C09144=1205.549,-72.595,-39.498,179.562,5.497,149.096
C09145=1205.554,-72.845,-39.488,179.559,5.497,149.096
C09146=1205.559,-73.095,-39.476,179.557,5.497,149.097
C09147=1205.565,-73.344,-39.465,179.555,5.497,149.098
C09148=1205.570,-73.594,-39.454,179.553,5.497,149.098
C09149=1205.574,-73.844,-39.443,179.550,5.496,149.099
C09150=1205.580,-74.093,-39.432,179.548,5.497,149.100
C09151=1205.585,-74.343,-39.421,179.545,5.496,149.100
C09152=1205.590,-74.593,-39.410,179.543,5.496,149.101
C09153=1205.596,-74.863,-39.398,179.540,5.496,149.102
C09154=1205.602,-75.134,-39.386,179.538,5.496,149.102
C09155=1205.608,-75.405,-39.373,179.535,5.495,149.103
C09156=1205.613,-75.675,-39.362,179.533,5.496,149.104
C09157=1205.619,-75.925,-39.351,179.530,5.495,149.105
C09158=1205.624,-76.174,-39.340,179.528,5.495,149.105
C09159=1205.629,-76.424,-39.329,179.526,5.495,149.106
C09160=1205.634,-76.674,-39.318,179.523,5.494,149.106
C09161=1205.640,-76.923,-39.307,179.521,5.495,149.107
C09162=1205.645,-77.174,-39.296,179.519,5.494,149.108
C09163=1205.650,-77.423,-39.285,179.516,5.495,149.109
C09164=1205.655,-77.673,-39.275,179.514,5.494,149.109
C09165=1205.661,-77.923,-39.263,179.512,5.494,149.110
C09166=1205.666,-78.172,-39.252,179.510,5.494,149.111
C09167=1205.671,-78.422,-39.241,179.507,5.493,149.111
C09168=1205.676,-78.672,-39.230,179.505,5.494,149.112
C09169=1205.681,-78.921,-39.220,179.502,5.493,149.113
C09170=1205.687,-79.171,-39.208,179.501,5.493,149.113
C09171=1205.692,-79.421,-39.198,179.498,5.493,149.114
C09172=1205.697,-79.670,-39.186,179.496,5.493,149.115
C09173=1205.702,-79.921,-39.176,179.493,5.493,149.115
C09174=1205.707,-80.169,-39.165,179.490,5.492,149.116
C09175=1205.712,-80.420,-39.154,179.489,5.492,149.116
C09176=1205.718,-80.669,-39.143,179.486,5.492,149.117
C09177=1205.723,-80.919,-39.132,179.484,5.492,149.118
C09178=1205.728,-81.169,-39.122,179.481,5.492,149.119
C09179=1205.733,-81.418,-39.111,179.479,5.492,149.119
C09180=1205.738,-81.669,-39.100,179.477,5.491,149.120
C09181=1205.744,-81.918,-39.089,179.475,5.492,149.120
C09182=1205.749,-82.168,-39.079,179.472,5.491,149.121
C09183=1205.755,-82.417,-39.067,179.470,5.491,149.122
C09184=1205.760,-82.667,-39.056,179.468,5.491,149.123
C09185=1205.765,-82.917,-39.046,179.465,5.490,149.123
C09186=1205.770,-83.166,-39.035,179.463,5.491,149.124
C09187=1205.775,-83.417,-39.024,179.461,5.490,149.124
C09188=1205.780,-83.666,-39.013,179.459,5.491,149.125
C09189=1205.785,-83.916,-39.003,179.456,5.490,149.126
C09190=1205.791,-84.165,-38.993,179.454,5.489,149.126
C09191=1205.796,-84.415,-38.981,179.452,5.490,149.127
C09192=1205.801,-84.665,-38.971,179.449,5.489,149.128
C09193=1205.806,-84.914,-38.960,179.447,5.490,149.129
C09194=1205.812,-85.164,-38.950,179.444,5.489,149.129
C09195=1205.817,-85.414,-38.939,179.443,5.489,149.130
C09196=1205.823,-85.663,-38.928,179.440,5.489,149.130
C09197=1205.828,-85.913,-38.917,179.438,5.489,149.131
C09198=1205.833,-86.163,-38.907,179.435,5.489,149.132
C09199=1205.838,-86.413,-38.895,179.433,5.489,149.133
C09200=1205.843,-86.662,-38.885,179.431,5.488,149.133
C09201=1205.848,-86.912,-38.875,179.428,5.488,149.134
C09202=1205.854,-87.162,-38.864,179.426,5.488,149.134
C09203=1205.859,-87.412,-38.853,179.423,5.488,149.135
C09204=1205.864,-87.661,-38.843,179.421,5.488,149.136
C09205=1205.869,-87.911,-38.832,179.419,5.487,149.136
C09206=1205.875,-88.160,-38.821,179.417,5.488,149.137
C09207=1205.880,-88.411,-38.811,179.414,5.487,149.138
C09208=1205.885,-88.660,-38.801,179.412,5.488,149.138
C09209=1205.890,-88.910,-38.790,179.410,5.487,149.139
C09210=1205.895,-89.159,-38.779,179.408,5.487,149.140
C09211=1205.900,-89.409,-38.769,179.405,5.487,149.140
C09212=1205.906,-89.659,-38.758,179.403,5.486,149.141
C09213=1205.911,-89.909,-38.748,179.401,5.487,149.142
C09214=1205.917,-90.159,-38.738,179.398,5.486,149.143
C09215=1205.921,-90.408,-38.726,179.396,5.486,149.143
C09216=1205.927,-90.658,-38.716,179.394,5.486,149.144
C09217=1205.932,-90.908,-38.706,179.392,5.486,149.144
C09218=1205.937,-91.157,-38.696,179.389,5.486,149.145
C09219=1205.942,-91.407,-38.686,179.387,5.486,149.146
C09220=1205.947,-91.657,-38.675,179.385,5.485,149.146
C09221=1205.953,-91.906,-38.664,179.383,5.486,149.147
C09222=1205.958,-92.156,-38.654,179.380,5.485,149.148
C09223=1205.963,-92.406,-38.643,179.378,5.486,149.148
C09224=1205.968,-92.656,-38.633,179.376,5.485,149.149
C09225=1205.974,-92.906,-38.623,179.374,5.485,149.150
C09226=1205.980,-93.155,-38.612,179.371,5.485,149.150
C09227=1205.985,-93.406,-38.602,179.368,5.485,149.151
C09228=1205.990,-93.654,-38.591,179.367,5.485,149.152
C09229=1205.995,-93.905,-38.580,179.364,5.484,149.152
C09230=1206.000,-94.154,-38.571,179.362,5.484,149.153
C09231=1206.005,-94.403,-38.561,179.359,5.484,149.154
C09232=1206.010,-94.654,-38.550,179.357,5.484,149.154
C09233=1206.016,-94.903,-38.540,179.355,5.484,149.155
C09234=1206.021,-95.154,-38.529,179.353,5.484,149.156
C09235=1206.026,-95.403,-38.519,179.350,5.484,149.156
C09236=1206.032,-95.653,-38.509,179.348,5.484,149.157
C09237=1206.037,-95.903,-38.498,179.346,5.483,149.158
C09238=1206.042,-96.152,-38.489,179.344,5.484,149.158
C09239=1206.048,-96.402,-38.478,179.341,5.483,149.159
C09240=1206.053,-96.652,-38.468,179.339,5.484,149.160
C09241=1206.058,-96.901,-38.458,179.337,5.483,149.160
C09242=1206.063,-97.152,-38.447,179.335,5.483,149.161
C09243=1206.069,-97.401,-38.437,179.332,5.483,149.162
C09244=1206.074,-97.650,-38.427,179.330,5.483,149.162
C09245=1206.079,-97.901,-38.417,179.328,5.482,149.163
C09246=1206.084,-98.150,-38.406,179.325,5.482,149.163
C09247=1206.090,-98.400,-38.396,179.323,5.482,149.164
C09248=1206.095,-98.650,-38.386,179.320,5.482,149.165
C09249=1206.100,-98.900,-38.375,179.319,5.482,149.165
C09250=1206.105,-99.149,-38.366,179.316,5.481,149.166
C09251=1206.110,-99.399,-38.355,179.314,5.482,149.167
C09252=1206.116,-99.649,-38.345,179.311,5.481,149.168
C09253=1206.121,-99.898,-38.335,179.309,5.482,149.168
C09254=1206.126,-100.148,-38.325,179.307,5.481,149.169
C09255=1206.131,-100.398,-38.315,179.305,5.481,149.169
C09256=1206.137,-100.647,-38.304,179.302,5.481,149.170
C09257=1206.142,-100.918,-38.294,179.300,5.481,149.171
C09258=1206.148,-101.190,-38.282,179.297,5.481,149.172
C09259=1206.154,-101.461,-38.271,179.295,5.480,149.172
C09260=1206.160,-101.733,-38.261,179.293,5.481,149.173
C09261=1206.164,-101.983,-38.251,179.291,5.480,149.173
C09262=1206.170,-102.232,-38.240,179.288,5.480,149.174
C09263=1206.175,-102.482,-38.230,179.286,5.480,149.175
C09264=1206.180,-102.731,-38.221,179.284,5.480,149.176
C09265=1206.185,-102.981,-38.210,179.281,5.480,149.176
C09266=1206.191,-103.231,-38.200,179.279,5.480,149.177
C09267=1206.196,-103.480,-38.190,179.277,5.480,149.178
C09268=1206.201,-103.731,-38.180,179.275,5.480,149.178
C09269=1206.207,-103.981,-38.170,179.272,5.479,149.179
C09270=1206.212,-104.230,-38.160,179.270,5.480,149.179
C09271=1206.217,-104.479,-38.150,179.268,5.479,149.180
C09272=1206.222,-104.730,-38.140,179.266,5.479,149.181
C09273=1206.228,-104.980,-38.130,179.263,5.479,149.181
C09274=1206.233,-105.229,-38.121,179.261,5.479,149.182
C09275=1206.238,-105.478,-38.110,179.259,5.479,149.183
C09276=1206.243,-105.729,-38.100,179.257,5.479,149.183
C09277=1206.248,-105.978,-38.090,179.254,5.478,149.184
C09278=1206.254,-106.228,-38.081,179.252,5.479,149.185
C09279=1206.260,-106.478,-38.071,179.250,5.478,149.185
C09280=1206.264,-106.728,-38.061,179.248,5.479,149.186
C09281=1206.270,-106.977,-38.050,179.245,5.478,149.187
C09282=1206.276,-107.227,-38.041,179.243,5.478,149.187
C09283=1206.280,-107.477,-38.031,179.241,5.478,149.188
C09284=1206.285,-107.727,-38.021,179.239,5.478,149.189
C09285=1206.290,-107.976,-38.011,179.236,5.477,149.189
C09286=1206.296,-108.226,-38.002,179.234,5.478,149.190
C09287=1206.302,-108.476,-37.991,179.232,5.477,149.191
C09288=1206.307,-108.725,-37.982,179.230,5.477,149.191
C09289=1206.312,-108.976,-37.972,179.227,5.477,149.192
C09290=1206.317,-109.225,-37.962,179.225,5.477,149.193
C09291=1206.322,-109.475,-37.952,179.222,5.477,149.193
C09292=1206.328,-109.724,-37.942,179.221,5.477,149.194
C09293=1206.333,-109.974,-37.933,179.218,5.477,149.194
C09294=1206.338,-110.224,-37.922,179.216,5.477,149.195
C09295=1206.343,-110.473,-37.913,179.214,5.476,149.196
C09296=1206.349,-110.724,-37.903,179.212,5.476,149.196
C09297=1206.355,-110.973,-37.893,179.209,5.476,149.197
C09298=1206.359,-111.222,-37.883,179.207,5.476,149.198
C09299=1206.365,-111.473,-37.874,179.205,5.476,149.198
C09300=1206.370,-111.722,-37.864,179.203,5.476,149.199
C09301=1206.376,-111.973,-37.854,179.200,5.476,149.200
C09302=1206.380,-112.222,-37.845,179.199,5.476,149.200
C09303=1206.386,-112.471,-37.835,179.196,5.475,149.201
C09304=1206.391,-112.721,-37.826,179.194,5.476,149.202
C09305=1206.396,-112.972,-37.815,179.192,5.475,149.202
C09306=1206.401,-113.221,-37.806,179.189,5.475,149.203
C09307=1206.407,-113.471,-37.796,179.187,5.475,149.204
C09308=1206.412,-113.720,-37.786,179.185,5.475,149.204
C09309=1206.418,-113.970,-37.777,179.182,5.474,149.205
C09310=1206.423,-114.220,-37.767,179.180,5.475,149.205
C09311=1206.428,-114.470,-37.758,179.178,5.475,149.206
C09312=1206.433,-114.720,-37.748,179.176,5.474,149.207
C09313=1206.439,-114.970,-37.738,179.174,5.475,149.207
C09314=1206.443,-115.219,-37.729,179.171,5.474,149.208
C09315=1206.449,-115.469,-37.719,179.169,5.475,149.209
C09316=1206.454,-115.718,-37.710,179.167,5.474,149.209
C09317=1206.460,-115.969,-37.700,179.165,5.474,149.210
C09318=1206.465,-116.218,-37.691,179.162,5.474,149.211
C09319=1206.471,-116.468,-37.681,179.161,5.474,149.211
C09320=1206.476,-116.717,-37.671,179.158,5.474,149.212
C09321=1206.481,-116.968,-37.662,179.156,5.474,149.213
C09322=1206.486,-117.217,-37.652,179.154,5.473,149.213
C09323=1206.492,-117.467,-37.642,179.152,5.474,149.214
C09324=1206.497,-117.717,-37.633,179.149,5.473,149.215
C09325=1206.502,-117.967,-37.624,179.147,5.473,149.215
C09326=1206.507,-118.216,-37.614,179.145,5.473,149.216
C09327=1206.513,-118.466,-37.605,179.143,5.473,149.217
C09328=1206.518,-118.716,-37.595,179.140,5.472,149.217
C09329=1206.523,-118.965,-37.586,179.138,5.473,149.218
C09330=1206.528,-119.215,-37.576,179.136,5.472,149.218
C09331=1206.534,-119.465,-37.567,179.134,5.473,149.219
C09332=1206.539,-119.715,-37.557,179.132,5.473,149.220
C09333=1206.544,-119.965,-37.547,179.129,5.472,149.220
C09334=1206.549,-120.215,-37.538,179.127,5.473,149.221
C09335=1206.554,-120.464,-37.529,179.125,5.472,149.222
C09336=1206.560,-120.714,-37.519,179.123,5.472,149.222
C09337=1206.565,-120.964,-37.510,179.120,5.472,149.223
C09338=1206.571,-121.213,-37.500,179.119,5.472,149.223
C09339=1206.576,-121.463,-37.491,179.116,5.472,149.224
C09340=1206.581,-121.713,-37.482,179.114,5.472,149.225
C09341=1206.587,-121.963,-37.472,179.112,5.471,149.225
C09342=1206.592,-122.213,-37.463,179.110,5.472,149.226
C09343=1206.597,-122.462,-37.454,179.107,5.471,149.227
C09344=1206.603,-122.712,-37.444,179.105,5.471,149.227
C09345=1206.608,-122.962,-37.435,179.103,5.471,149.228
C09346=1206.613,-123.211,-37.426,179.101,5.471,149.229
C09347=1206.619,-123.461,-37.416,179.099,5.471,149.229
C09348=1206.624,-123.711,-37.407,179.096,5.471,149.230
C09349=1206.629,-123.960,-37.398,179.094,5.471,149.231
C09350=1206.635,-124.210,-37.388,179.092,5.470,149.231
C09351=1206.640,-124.460,-37.379,179.090,5.471,149.232
C09352=1206.645,-124.710,-37.370,179.087,5.470,149.233
C09353=1206.650,-124.959,-37.361,179.086,5.470,149.233
C09354=1206.656,-125.210,-37.351,179.083,5.470,149.234
C09355=1206.661,-125.459,-37.342,179.081,5.470,149.234
C09356=1206.666,-125.709,-37.333,179.079,5.470,149.235
C09357=1206.672,-125.959,-37.323,179.077,5.470,149.236
C09358=1206.677,-126.209,-37.314,179.074,5.469,149.236
C09359=1206.682,-126.459,-37.305,179.072,5.470,149.237
C09360=1206.687,-126.708,-37.296,179.070,5.470,149.238
C09361=1206.266,-126.720,-37.333,179.066,5.473,149.239
C09362=1206.261,-126.470,-37.342,179.068,5.473,149.239
C09363=1206.255,-126.220,-37.352,179.070,5.473,149.238
C09364=1206.250,-125.970,-37.361,179.073,5.473,149.238
C09365=1206.245,-125.721,-37.370,179.074,5.473,149.237
C09366=1206.239,-125.470,-37.380,179.077,5.474,149.236
C09367=1206.234,-125.221,-37.389,179.079,5.473,149.236
C09368=1206.228,-124.971,-37.398,179.081,5.474,149.235
C09369=1206.224,-124.722,-37.407,179.083,5.474,149.234
C09370=1206.218,-124.471,-37.417,179.086,5.474,149.234
C09371=1206.213,-124.222,-37.426,179.088,5.474,149.233
C09372=1206.208,-123.972,-37.435,179.090,5.474,149.233
C09373=1206.202,-123.722,-37.445,179.092,5.474,149.232
C09374=1206.197,-123.472,-37.454,179.095,5.475,149.231
C09375=1206.192,-123.223,-37.463,179.097,5.474,149.231
C09376=1206.186,-122.973,-37.473,179.099,5.474,149.230
C09377=1206.181,-122.723,-37.482,179.101,5.475,149.229
C09378=1206.176,-122.474,-37.491,179.103,5.474,149.229
C09379=1206.170,-122.223,-37.501,179.106,5.475,149.228
C09380=1206.165,-121.973,-37.510,179.107,5.475,149.227
C09381=1206.160,-121.724,-37.520,179.110,5.475,149.227
C09382=1206.155,-121.474,-37.529,179.112,5.475,149.226
C09383=1206.149,-121.224,-37.538,179.114,5.476,149.226
C09384=1206.145,-120.975,-37.548,179.116,5.475,149.225
C09385=1206.139,-120.724,-37.557,179.119,5.476,149.224
C09386=1206.133,-120.475,-37.566,179.121,5.476,149.224
C09387=1206.128,-120.225,-37.576,179.123,5.476,149.223
C09388=1206.123,-119.975,-37.585,179.125,5.476,149.222
C09389=1206.118,-119.726,-37.595,179.128,5.476,149.222
C09390=1206.112,-119.476,-37.604,179.130,5.476,149.221
C09391=1206.107,-119.226,-37.613,179.132,5.476,149.220
C09392=1206.102,-118.977,-37.623,179.134,5.476,149.220
C09393=1206.096,-118.727,-37.632,179.136,5.476,149.219
C09394=1206.091,-118.477,-37.642,179.139,5.476,149.218
C09395=1206.085,-118.227,-37.651,179.140,5.476,149.218
C09396=1206.081,-117.977,-37.661,179.143,5.477,149.217
C09397=1206.075,-117.727,-37.671,179.145,5.476,149.216
C09398=1206.070,-117.478,-37.680,179.147,5.477,149.216
C09399=1206.065,-117.228,-37.689,179.149,5.477,149.215
C09400=1206.059,-116.978,-37.700,179.152,5.477,149.215
C09401=1206.054,-116.729,-37.708,179.154,5.477,149.214
C09402=1206.049,-116.479,-37.719,179.156,5.478,149.213
C09403=1206.044,-116.229,-37.728,179.158,5.477,149.213
C09404=1206.038,-115.980,-37.738,179.161,5.478,149.212
C09405=1206.033,-115.729,-37.747,179.163,5.478,149.211
C09406=1206.028,-115.480,-37.757,179.165,5.478,149.211
C09407=1206.023,-115.230,-37.766,179.167,5.478,149.210
C09408=1206.017,-114.980,-37.776,179.170,5.478,149.209
C09409=1206.012,-114.730,-37.785,179.172,5.478,149.209
C09410=1206.007,-114.481,-37.795,179.174,5.478,149.208
C09411=1206.001,-114.231,-37.804,179.176,5.478,149.208
C09412=1205.996,-113.982,-37.814,179.179,5.479,149.207
C09413=1205.991,-113.731,-37.824,179.181,5.478,149.206
C09414=1205.985,-113.481,-37.834,179.183,5.478,149.205
C09415=1205.980,-113.231,-37.843,179.185,5.479,149.205
C09416=1205.975,-112.982,-37.853,179.187,5.478,149.204
C09417=1205.970,-112.733,-37.863,179.190,5.479,149.204
C09418=1205.964,-112.482,-37.872,179.191,5.479,149.203
C09419=1205.959,-112.233,-37.882,179.194,5.479,149.202
C09420=1205.954,-111.982,-37.892,179.196,5.479,149.202
C09421=1205.949,-111.733,-37.901,179.198,5.480,149.201
C09422=1205.943,-111.484,-37.912,179.200,5.479,149.200
C09423=1205.938,-111.234,-37.920,179.203,5.480,149.200
C09424=1205.932,-110.984,-37.931,179.205,5.479,149.199
C09425=1205.928,-110.735,-37.940,179.207,5.480,149.198
C09426=1205.922,-110.484,-37.950,179.209,5.480,149.198
C09427=1205.917,-110.235,-37.960,179.212,5.480,149.197
C09428=1205.912,-109.985,-37.970,179.214,5.480,149.197
C09429=1205.906,-109.735,-37.979,179.216,5.480,149.196
C09430=1205.901,-109.486,-37.989,179.219,5.480,149.195
C09431=1205.896,-109.236,-38.000,179.221,5.480,149.194
C09432=1205.891,-108.986,-38.009,179.223,5.481,149.194
C09433=1205.885,-108.736,-38.019,179.225,5.481,149.193
C09434=1205.880,-108.487,-38.029,179.228,5.481,149.193
C09435=1205.874,-108.237,-38.038,179.230,5.481,149.192
C09436=1205.869,-107.987,-38.048,179.232,5.481,149.191
C09437=1205.864,-107.737,-38.059,179.235,5.481,149.191
C09438=1205.859,-107.488,-38.068,179.237,5.481,149.190
C09439=1205.853,-107.238,-38.078,179.239,5.482,149.189
C09440=1205.848,-106.989,-38.087,179.241,5.481,149.189
C09441=1205.843,-106.738,-38.098,179.244,5.482,149.188
C09442=1205.838,-106.489,-38.108,179.246,5.481,149.187
C09443=1205.832,-106.239,-38.117,179.248,5.482,149.187
C09444=1205.827,-105.989,-38.127,179.250,5.482,149.186
C09445=1205.822,-105.739,-38.138,179.253,5.482,149.185
C09446=1205.817,-105.490,-38.147,179.254,5.482,149.185
C09447=1205.811,-105.240,-38.157,179.257,5.483,149.184
C09448=1205.806,-104.990,-38.167,179.259,5.482,149.183
C09449=1205.801,-104.740,-38.177,179.262,5.483,149.183
C09450=1205.796,-104.491,-38.187,179.263,5.483,149.182
C09451=1205.790,-104.241,-38.198,179.266,5.483,149.182
C09452=1205.786,-103.991,-38.207,179.268,5.483,149.181
C09453=1205.780,-103.741,-38.217,179.271,5.483,149.180
C09454=1205.774,-103.491,-38.227,179.272,5.483,149.180
C09455=1205.769,-103.242,-38.237,179.275,5.484,149.179
C09456=1205.764,-102.992,-38.247,179.277,5.483,149.178
C09457=1205.759,-102.742,-38.258,179.280,5.484,149.177
C09458=1205.754,-102.493,-38.267,179.281,5.484,149.177
C09459=1205.749,-102.242,-38.277,179.284,5.484,149.176
C09460=1205.743,-101.993,-38.287,179.286,5.484,149.176
C09461=1205.737,-101.743,-38.298,179.289,5.484,149.175
C09462=1205.732,-101.472,-38.308,179.291,5.484,149.174
C09463=1205.727,-101.201,-38.319,179.294,5.484,149.173
C09464=1205.721,-100.930,-38.331,179.296,5.484,149.173
C09465=1205.715,-100.658,-38.342,179.298,5.484,149.172
C09466=1205.710,-100.408,-38.351,179.300,5.485,149.172
C09467=1205.705,-100.158,-38.362,179.303,5.484,149.171
C09468=1205.699,-99.909,-38.372,179.305,5.485,149.170
C09469=1205.694,-99.659,-38.381,179.307,5.484,149.169
C09470=1205.689,-99.409,-38.392,179.310,5.485,149.169
C09471=1205.683,-99.160,-38.402,179.312,5.486,149.168
C09472=1205.678,-98.910,-38.412,179.314,5.485,149.167
C09473=1205.674,-98.660,-38.422,179.317,5.486,149.167
C09474=1205.668,-98.410,-38.433,179.319,5.486,149.166
C09475=1205.662,-98.161,-38.443,179.321,5.486,149.166
C09476=1205.657,-97.911,-38.453,179.323,5.486,149.165
C09477=1205.652,-97.661,-38.464,179.326,5.486,149.164
C09478=1205.647,-97.412,-38.473,179.328,5.486,149.164
C09479=1205.642,-97.162,-38.484,179.330,5.487,149.163
C09480=1205.636,-96.912,-38.494,179.332,5.486,149.162
C09481=1205.631,-96.663,-38.504,179.335,5.487,149.162
C09482=1205.626,-96.412,-38.515,179.337,5.487,149.161
C09483=1205.620,-96.163,-38.525,179.339,5.487,149.160
C09484=1205.615,-95.913,-38.536,179.341,5.487,149.160
C09485=1205.610,-95.663,-38.545,179.344,5.487,149.159
C09486=1205.605,-95.414,-38.555,179.346,5.487,149.158
C09487=1205.600,-95.164,-38.566,179.348,5.488,149.158
C09488=1205.594,-94.914,-38.576,179.350,5.487,149.157
C09489=1205.588,-94.664,-38.586,179.353,5.488,149.156
C09490=1205.583,-94.414,-38.597,179.355,5.488,149.156
C09491=1205.578,-94.165,-38.608,179.357,5.488,149.155
C09492=1205.574,-93.915,-38.618,179.359,5.488,149.154
C09493=1205.568,-93.666,-38.628,179.362,5.488,149.154
C09494=1205.563,-93.416,-38.638,179.365,5.488,149.153
C09495=1205.558,-93.166,-38.649,179.366,5.488,149.152
C09496=1205.552,-92.916,-38.659,179.369,5.489,149.152
C09497=1205.547,-92.666,-38.670,179.371,5.489,149.151
C09498=1205.542,-92.417,-38.680,179.374,5.489,149.150
C09499=1205.537,-92.166,-38.690,179.375,5.489,149.150
C09500=1205.531,-91.918,-38.701,179.378,5.489,149.149
C09501=1205.526,-91.668,-38.712,179.380,5.489,149.148
C09502=1205.521,-91.418,-38.722,179.383,5.489,149.148
C09503=1205.515,-91.168,-38.732,179.385,5.489,149.147
C09504=1205.510,-90.918,-38.743,179.387,5.490,149.147
C09505=1205.505,-90.669,-38.753,179.389,5.489,149.146
C09506=1205.501,-90.419,-38.764,179.392,5.490,149.145
C09507=1205.495,-90.170,-38.774,179.395,5.490,149.144
C09508=1205.489,-89.920,-38.784,179.396,5.490,149.144
C09509=1205.484,-89.670,-38.795,179.399,5.491,149.143
C09510=1205.479,-89.421,-38.806,179.401,5.490,149.142
C09511=1205.474,-89.171,-38.816,179.404,5.491,149.142
C09512=1205.468,-88.921,-38.826,179.406,5.490,149.141
C09513=1205.463,-88.671,-38.837,179.408,5.491,149.141
C09514=1205.458,-88.421,-38.847,179.410,5.491,149.140
C09515=1205.453,-88.172,-38.859,179.413,5.491,149.139
C09516=1205.448,-87.922,-38.869,179.415,5.491,149.138
C09517=1205.443,-87.672,-38.879,179.417,5.492,149.138
C09518=1205.437,-87.422,-38.890,179.419,5.491,149.137
C09519=1205.432,-87.173,-38.901,179.422,5.492,149.137
C09520=1205.427,-86.923,-38.911,179.424,5.492,149.136
C09521=1205.422,-86.673,-38.922,179.426,5.492,149.135
C09522=1205.416,-86.424,-38.933,179.429,5.493,149.135
C09523=1205.411,-86.174,-38.943,179.431,5.492,149.134
C09524=1205.406,-85.924,-38.953,179.433,5.493,149.133
C09525=1205.401,-85.675,-38.965,179.435,5.492,149.133
C09526=1205.395,-85.425,-38.975,179.438,5.493,149.132
C09527=1205.390,-85.175,-38.985,179.440,5.493,149.131
C09528=1205.384,-84.926,-38.997,179.442,5.493,149.131
C09529=1205.379,-84.675,-39.008,179.445,5.494,149.130
C09530=1205.374,-84.426,-39.018,179.447,5.493,149.129
C09531=1205.369,-84.176,-39.029,179.450,5.494,149.128
C09532=1205.364,-83.927,-39.039,179.451,5.494,149.128
C09533=1205.359,-83.676,-39.050,179.454,5.494,149.127
C09534=1205.354,-83.427,-39.061,179.456,5.494,149.127
C09535=1205.348,-83.177,-39.071,179.459,5.494,149.126
C09536=1205.344,-82.928,-39.083,179.461,5.494,149.125
C09537=1205.338,-82.678,-39.093,179.463,5.495,149.125
C09538=1205.333,-82.428,-39.103,179.466,5.495,149.124
C09539=1205.328,-82.179,-39.114,179.468,5.495,149.123
C09540=1205.322,-81.928,-39.125,179.471,5.495,149.123
C09541=1205.317,-81.679,-39.136,179.473,5.495,149.122
C09542=1205.312,-81.429,-39.147,179.475,5.496,149.121
C09543=1205.307,-81.179,-39.158,179.477,5.495,149.121
C09544=1205.301,-80.930,-39.168,179.480,5.496,149.120
C09545=1205.296,-80.680,-39.179,179.482,5.495,149.119
C09546=1205.291,-80.431,-39.190,179.484,5.496,149.119
C09547=1205.285,-80.180,-39.201,179.487,5.496,149.118
C09548=1205.280,-79.931,-39.212,179.489,5.496,149.117
C09549=1205.275,-79.681,-39.223,179.491,5.497,149.117
C09550=1205.270,-79.431,-39.234,179.493,5.496,149.116
C09551=1205.265,-79.182,-39.244,179.496,5.497,149.115
C09552=1205.260,-78.932,-39.255,179.498,5.497,149.115
C09553=1205.254,-78.682,-39.266,179.500,5.497,149.114
C09554=1205.249,-78.433,-39.277,179.503,5.497,149.113
C09555=1205.244,-78.183,-39.288,179.505,5.497,149.113
C09556=1205.239,-77.934,-39.299,179.508,5.498,149.112
C09557=1205.234,-77.684,-39.310,179.510,5.497,149.111
C09558=1205.228,-77.434,-39.321,179.512,5.498,149.111
C09559=1205.223,-77.184,-39.332,179.514,5.498,149.110
C09560=1205.218,-76.934,-39.343,179.517,5.498,149.109
C09561=1205.213,-76.685,-39.354,179.519,5.499,149.109
C09562=1205.207,-76.435,-39.365,179.522,5.498,149.108
C09563=1205.202,-76.185,-39.376,179.524,5.499,149.107
C09564=1205.197,-75.936,-39.387,179.526,5.499,149.107
C09565=1205.192,-75.686,-39.398,179.528,5.499,149.106
C09566=1205.186,-75.416,-39.410,179.531,5.499,149.105
C09567=1205.180,-75.145,-39.422,179.533,5.499,149.105
C09568=1205.175,-74.874,-39.434,179.536,5.500,149.104
C09569=1205.169,-74.604,-39.446,179.539,5.500,149.103
C09570=1205.164,-74.354,-39.457,179.541,5.500,149.102
C09571=1205.159,-74.104,-39.468,179.543,5.500,149.102
C09572=1205.153,-73.855,-39.479,179.546,5.500,149.101
C09573=1205.148,-73.605,-39.491,179.548,5.500,149.100
C09574=1205.143,-73.354,-39.501,179.550,5.501,149.100
C09575=1205.138,-73.106,-39.512,179.552,5.501,149.099
C09576=1205.132,-72.856,-39.524,179.555,5.501,149.098
C09577=1205.127,-72.605,-39.535,179.557,5.501,149.098
C09578=1205.122,-72.356,-39.546,179.560,5.501,149.097
C09579=1205.117,-72.107,-39.558,179.562,5.502,149.097
C09580=1205.112,-71.856,-39.568,179.564,5.502,149.096
C09581=1205.107,-71.607,-39.579,179.567,5.502,149.095
C09582=1205.101,-71.357,-39.591,179.569,5.502,149.094
C09583=1205.096,-71.108,-39.602,179.571,5.502,149.094
C09584=1205.091,-70.858,-39.613,179.574,5.502,149.093
C09585=1205.085,-70.608,-39.624,179.576,5.502,149.093
C09586=1205.080,-70.359,-39.636,179.578,5.503,149.092
C09587=1205.075,-70.108,-39.646,179.581,5.503,149.091
C09588=1205.069,-69.859,-39.658,179.583,5.503,149.090
C09589=1205.065,-69.610,-39.669,179.586,5.503,149.090
C09590=1205.060,-69.360,-39.680,179.588,5.503,149.089
C09591=1205.055,-69.110,-39.692,179.590,5.504,149.088
C09592=1205.049,-68.860,-39.702,179.592,5.504,149.088
C09593=1205.044,-68.611,-39.714,179.595,5.504,149.087
C09594=1205.039,-68.361,-39.726,179.598,5.504,149.086
C09595=1205.034,-68.111,-39.737,179.600,5.504,149.086
C09596=1205.028,-67.862,-39.748,179.602,5.504,149.085
C09597=1205.023,-67.612,-39.759,179.604,5.505,149.084
C09598=1205.018,-67.362,-39.771,179.607,5.505,149.084
C09599=1205.013,-67.112,-39.782,179.609,5.505,149.083
C09600=1205.008,-66.863,-39.793,179.611,5.505,149.082
C09601=1205.002,-66.613,-39.805,179.614,5.505,149.082
C09602=1204.998,-66.364,-39.816,179.616,5.505,149.081
C09603=1204.992,-66.114,-39.828,179.618,5.506,149.080
C09604=1204.987,-65.864,-39.838,179.621,5.506,149.080
C09605=1204.981,-65.614,-39.850,179.623,5.506,149.079
C09606=1204.976,-65.365,-39.861,179.626,5.506,149.078
C09607=1204.971,-65.115,-39.873,179.628,5.506,149.078
C09608=1204.966,-64.865,-39.885,179.630,5.507,149.077
C09609=1204.960,-64.616,-39.896,179.633,5.507,149.076
C09610=1204.956,-64.366,-39.907,179.635,5.507,149.076
C09611=1204.950,-64.116,-39.919,179.637,5.507,149.075
C09612=1204.945,-63.867,-39.931,179.639,5.507,149.074
C09613=1204.940,-63.617,-39.943,179.642,5.508,149.074
C09614=1204.935,-63.368,-39.953,179.645,5.508,149.073
C09615=1204.929,-63.117,-39.965,179.646,5.508,149.072
C09616=1204.924,-62.868,-39.976,179.649,5.508,149.072
C09617=1204.919,-62.618,-39.988,179.652,5.509,149.071
C09618=1204.914,-62.368,-39.999,179.654,5.509,149.070
C09619=1204.909,-62.118,-40.011,179.656,5.509,149.070
C09620=1204.903,-61.869,-40.022,179.659,5.509,149.069
C09621=1204.898,-61.619,-40.034,179.661,5.509,149.068
C09622=1204.893,-61.370,-40.045,179.663,5.510,149.068
C09623=1204.888,-61.120,-40.057,179.665,5.510,149.067
C09624=1204.883,-60.870,-40.068,179.668,5.510,149.066
C09625=1204.878,-60.620,-40.080,179.671,5.510,149.066
C09626=1204.873,-60.371,-40.091,179.673,5.510,149.065
C09627=1204.867,-60.121,-40.103,179.676,5.511,149.064
C09628=1204.863,-59.872,-40.115,179.677,5.511,149.064
C09629=1204.857,-59.622,-40.127,179.680,5.511,149.063
C09630=1204.852,-59.372,-40.139,179.683,5.511,149.062
C09631=1204.847,-59.123,-40.150,179.685,5.511,149.062
C09632=1204.842,-58.873,-40.162,179.687,5.512,149.061
C09633=1204.837,-58.623,-40.173,179.690,5.512,149.060
C09634=1204.831,-58.374,-40.185,179.692,5.512,149.060
C09635=1204.826,-58.124,-40.197,179.694,5.512,149.059
C09636=1204.821,-57.874,-40.208,179.696,5.512,149.058
C09637=1204.815,-57.625,-40.220,179.699,5.513,149.058
C09638=1204.811,-57.375,-40.231,179.702,5.513,149.057
C09639=1204.806,-57.126,-40.244,179.704,5.513,149.056
C09640=1204.800,-56.876,-40.256,179.706,5.513,149.056
C09641=1204.796,-56.626,-40.267,179.709,5.514,149.055
C09642=1204.790,-56.376,-40.279,179.711,5.514,149.054
C09643=1204.785,-56.126,-40.291,179.713,5.514,149.054
C09644=1204.780,-55.877,-40.302,179.716,5.514,149.053
C09645=1204.774,-55.627,-40.313,179.718,5.514,149.052
C09646=1204.770,-55.378,-40.325,179.721,5.515,149.052
C09647=1204.764,-55.128,-40.337,179.723,5.515,149.051
C09648=1204.759,-54.878,-40.349,179.725,5.515,149.050
C09649=1204.754,-54.629,-40.360,179.728,5.516,149.050
C09650=1204.749,-54.379,-40.372,179.730,5.515,149.049
C09651=1204.743,-54.130,-40.385,179.732,5.516,149.048
C09652=1204.738,-53.880,-40.397,179.735,5.516,149.048
C09653=1204.733,-53.630,-40.408,179.737,5.516,149.047
C09654=1204.728,-53.380,-40.420,179.740,5.516,149.046
C09655=1204.723,-53.131,-40.433,179.742,5.517,149.046
C09656=1204.718,-52.881,-40.444,179.744,5.517,149.045
C09657=1204.713,-52.631,-40.456,179.747,5.517,149.044
C09658=1204.707,-52.381,-40.468,179.749,5.518,149.044
C09659=1204.703,-52.132,-40.480,179.751,5.517,149.043
C09660=1204.697,-51.882,-40.492,179.754,5.518,149.042
C09661=1204.692,-51.632,-40.503,179.757,5.518,149.041
C09662=1204.687,-51.383,-40.516,179.758,5.518,149.041
C09663=1204.682,-51.133,-40.527,179.761,5.519,149.040
C09664=1204.677,-50.883,-40.539,179.764,5.519,149.040
C09665=1204.671,-50.634,-40.551,179.766,5.519,149.039
C09666=1204.666,-50.384,-40.564,179.768,5.519,149.038
C09667=1204.661,-50.134,-40.576,179.771,5.520,149.037
C09668=1204.656,-49.885,-40.587,179.773,5.519,149.037
C09669=1204.651,-49.635,-40.599,179.775,5.520,149.036
C09670=1204.645,-49.366,-40.612,179.779,5.520,149.035
C09671=1204.640,-49.095,-40.625,179.781,5.520,149.035
C09672=1204.634,-48.825,-40.638,179.783,5.520,149.034
C09673=1204.628,-48.555,-40.651,179.786,5.521,149.033
C09674=1204.623,-48.306,-40.663,179.789,5.521,149.033
C09675=1204.618,-48.056,-40.675,179.790,5.521,149.032
C09676=1204.613,-47.807,-40.688,179.793,5.522,149.031
C09677=1204.607,-47.557,-40.700,179.796,5.522,149.031
C09678=1204.602,-47.307,-40.711,179.798,5.522,149.030
C09679=1204.597,-47.058,-40.724,179.800,5.522,149.029
C09680=1204.592,-46.808,-40.735,179.803,5.523,149.029
C09681=1204.587,-46.559,-40.748,179.805,5.522,149.028
C09682=1204.582,-46.309,-40.760,179.808,5.523,149.027
C09683=1204.577,-46.058,-40.772,179.810,5.524,149.027
C09684=1204.572,-45.809,-40.785,179.812,5.523,149.026
C09685=1204.566,-45.559,-40.797,179.815,5.524,149.025
C09686=1204.561,-45.309,-40.809,179.817,5.524,149.025
C09687=1204.556,-45.060,-40.820,179.819,5.524,149.024
C09688=1204.551,-44.811,-40.833,179.822,5.524,149.023
C09689=1204.546,-44.561,-40.845,179.825,5.525,149.022
C09690=1204.541,-44.311,-40.858,179.827,5.526,149.022
C09691=1204.535,-44.061,-40.869,179.829,5.525,149.021
C09692=1204.530,-43.812,-40.882,179.832,5.526,149.021
C09693=1204.525,-43.562,-40.894,179.834,5.526,149.020
C09694=1204.520,-43.313,-40.907,179.836,5.526,149.019
C09695=1204.514,-43.063,-40.918,179.839,5.526,149.018
C09696=1204.510,-42.813,-40.931,179.842,5.527,149.018
C09697=1204.505,-42.563,-40.944,179.843,5.527,149.017
C09698=1204.499,-42.314,-40.956,179.846,5.527,149.017
C09699=1204.495,-42.065,-40.968,179.849,5.528,149.016
C09700=1204.489,-41.815,-40.980,179.851,5.527,149.015
C09701=1204.484,-41.565,-40.992,179.853,5.528,149.014
C09702=1204.479,-41.315,-41.004,179.856,5.528,149.014
C09703=1204.474,-41.066,-41.017,179.858,5.528,149.013
C09704=1204.468,-40.817,-41.029,179.861,5.528,149.012
C09705=1204.464,-40.566,-41.042,179.863,5.529,149.012
C09706=1204.459,-40.317,-41.054,179.866,5.530,149.011
C09707=1204.453,-40.067,-41.066,179.868,5.529,149.011
C09708=1204.448,-39.818,-41.079,179.870,5.530,149.010
C09709=1204.443,-39.568,-41.091,179.873,5.530,149.009
C09710=1204.437,-39.318,-41.103,179.875,5.530,149.008
C09711=1204.432,-39.069,-41.116,179.878,5.530,149.008
C09712=1204.428,-38.819,-41.129,179.880,5.531,149.007
C09713=1204.422,-38.569,-41.141,179.882,5.531,149.007
C09714=1204.417,-38.320,-41.153,179.885,5.531,149.006
C09715=1204.412,-38.070,-41.166,179.887,5.532,149.005
C09716=1204.407,-37.820,-41.178,179.890,5.532,149.004
C09717=1204.402,-37.571,-41.190,179.892,5.532,149.004
C09718=1204.397,-37.321,-41.203,179.895,5.532,149.003
C09719=1204.392,-37.072,-41.216,179.897,5.533,149.003
C09720=1204.386,-36.821,-41.228,179.899,5.533,149.002
C09721=1204.381,-36.572,-41.241,179.902,5.533,149.001
C09722=1204.375,-36.323,-41.254,179.904,5.534,149.000
C09723=1204.370,-36.074,-41.266,179.906,5.534,149.000
C09724=1204.366,-35.823,-41.279,179.909,5.534,148.999
C09725=1204.360,-35.574,-41.291,179.912,5.534,148.998
C09726=1204.355,-35.324,-41.304,179.914,5.535,148.998
C09727=1204.350,-35.075,-41.316,179.916,5.535,148.997
C09728=1204.345,-34.824,-41.329,179.919,5.535,148.996
C09729=1204.340,-34.575,-41.341,179.921,5.536,148.996
C09730=1204.335,-34.326,-41.354,179.923,5.536,148.995
C09731=1204.329,-34.076,-41.367,179.926,5.536,148.994
C09732=1204.324,-33.827,-41.380,179.929,5.537,148.994
C09733=1204.319,-33.576,-41.392,179.931,5.537,148.993
C09734=1204.314,-33.327,-41.404,179.933,5.537,148.993
C09735=1204.309,-33.077,-41.417,179.936,5.538,148.992
C09736=1204.304,-32.828,-41.430,179.938,5.538,148.991
C09737=1204.299,-32.578,-41.443,179.940,5.538,148.990
C09738=1204.294,-32.329,-41.456,179.943,5.538,148.990
C09739=1204.288,-32.079,-41.468,179.946,5.539,148.989
C09740=1204.283,-31.829,-41.480,179.948,5.539,148.988
C09741=1204.278,-31.579,-41.493,179.950,5.539,148.988
C09742=1204.273,-31.330,-41.506,179.953,5.540,148.987
C09743=1204.268,-31.081,-41.518,179.955,5.540,148.986
C09744=1204.262,-30.831,-41.532,179.958,5.540,148.986
C09745=1204.258,-30.581,-41.545,179.960,5.540,148.985
C09746=1204.253,-30.332,-41.557,179.963,5.541,148.984
C09747=1204.248,-30.082,-41.570,179.965,5.541,148.984
C09748=1204.242,-29.833,-41.582,179.968,5.542,148.983
C09749=1204.237,-29.583,-41.596,179.970,5.542,148.983
C09750=1204.232,-29.333,-41.609,179.972,5.542,148.982
C09751=1204.227,-29.083,-41.620,179.975,5.543,148.981
C09752=1204.222,-28.833,-41.633,179.977,5.542,148.980
C09753=1204.217,-28.584,-41.646,179.980,5.543,148.980
C09754=1204.211,-28.334,-41.659,179.982,5.543,148.979
C09755=1204.207,-28.084,-41.672,179.985,5.544,148.978
C09756=1204.201,-27.835,-41.685,179.987,5.543,148.978
C09757=1204.196,-27.586,-41.697,179.989,5.544,148.977
C09758=1204.191,-27.335,-41.711,179.992,5.545,148.976
C09759=1204.186,-27.086,-41.724,179.995,5.545,148.976
C09760=1204.181,-26.837,-41.736,179.997,5.545,148.975
C09761=1204.176,-26.587,-41.749,179.999,5.545,148.974
C09762=1204.171,-26.338,-41.763,-179.998,5.546,148.974
C09763=1204.166,-26.088,-41.776,-179.995,5.546,148.973
C09764=1204.161,-25.838,-41.789,-179.993,5.546,148.972
C09765=1204.155,-25.589,-41.802,-179.991,5.547,148.972
C09766=1204.150,-25.340,-41.814,-179.988,5.547,148.971
C09767=1204.146,-25.089,-41.827,-179.986,5.548,148.970
C09768=1204.140,-24.840,-41.840,-179.984,5.547,148.970
C09769=1204.135,-24.591,-41.853,-179.981,5.548,148.969
C09770=1204.130,-24.341,-41.866,-179.978,5.548,148.968
C09771=1204.125,-24.091,-41.879,-179.976,5.549,148.968
C09772=1204.119,-23.842,-41.892,-179.974,5.549,148.967
C09773=1204.115,-23.592,-41.905,-179.972,5.549,148.966
C09774=1204.109,-23.323,-41.920,-179.969,5.550,148.966
C09775=1204.104,-23.053,-41.933,-179.966,5.550,148.965
C09776=1204.098,-22.783,-41.947,-179.963,5.550,148.964
C09777=1204.093,-22.514,-41.962,-179.960,5.551,148.963
C09778=1204.087,-22.264,-41.975,-179.958,5.551,148.963
C09779=1204.082,-22.015,-41.988,-179.956,5.551,148.962
C09780=1204.077,-21.765,-42.001,-179.953,5.552,148.962
C09781=1204.072,-21.515,-42.014,-179.951,5.552,148.961
C09782=1204.067,-21.265,-42.027,-179.948,5.553,148.960
C09783=1204.062,-21.016,-42.041,-179.946,5.552,148.960
C09784=1204.057,-20.767,-42.053,-179.943,5.553,148.959
C09785=1204.051,-20.517,-42.067,-179.941,5.553,148.958
C09786=1204.046,-20.267,-42.079,-179.939,5.554,148.958
C09787=1204.042,-20.018,-42.093,-179.937,5.554,148.957
C09788=1204.036,-19.768,-42.106,-179.934,5.554,148.956
C09789=1204.031,-19.519,-42.119,-179.931,5.555,148.956
C09790=1204.026,-19.269,-42.133,-179.929,5.555,148.955
C09791=1204.021,-19.020,-42.146,-179.926,5.556,148.954
C09792=1204.016,-18.770,-42.159,-179.924,5.556,148.953
C09793=1204.010,-18.520,-42.172,-179.921,5.556,148.953
C09794=1204.006,-18.270,-42.185,-179.919,5.557,148.952
C09795=1204.000,-18.021,-42.199,-179.916,5.557,148.952
C09796=1203.996,-17.771,-42.212,-179.914,5.557,148.951
C09797=1203.990,-17.522,-42.225,-179.912,5.557,148.950
C09798=1203.985,-17.273,-42.238,-179.909,5.558,148.950
C09799=1203.980,-17.023,-42.252,-179.906,5.558,148.949
C09800=1203.975,-16.773,-42.265,-179.904,5.559,148.948
C09801=1203.970,-16.524,-42.279,-179.902,5.559,148.948
C09802=1203.965,-16.274,-42.291,-179.899,5.559,148.947
C09803=1203.959,-16.024,-42.305,-179.897,5.560,148.946
C09804=1203.955,-15.775,-42.318,-179.894,5.560,148.946
C09805=1203.949,-15.525,-42.332,-179.891,5.561,148.945
C09806=1203.944,-15.276,-42.344,-179.889,5.561,148.944
C09807=1203.939,-15.026,-42.359,-179.887,5.561,148.944
C09808=1203.934,-14.777,-42.371,-179.884,5.562,148.943
C09809=1203.929,-14.527,-42.386,-179.882,5.562,148.942
C09810=1203.923,-14.277,-42.399,-179.880,5.562,148.942
C09811=1203.919,-14.028,-42.412,-179.877,5.563,148.941
C09812=1203.913,-13.778,-42.426,-179.874,5.563,148.940
C09813=1203.909,-13.528,-42.439,-179.872,5.564,148.940
C09814=1203.903,-13.279,-42.453,-179.869,5.564,148.939
C09815=1203.899,-13.029,-42.465,-179.867,5.564,148.938
C09816=1203.893,-12.780,-42.479,-179.865,5.565,148.938
C09817=1203.888,-12.530,-42.493,-179.862,5.565,148.937
C09818=1203.884,-12.280,-42.507,-179.860,5.566,148.936
C09819=1203.878,-12.031,-42.520,-179.857,5.566,148.936
C09820=1203.874,-11.781,-42.534,-179.855,5.566,148.935
C09821=1203.868,-11.532,-42.547,-179.852,5.566,148.934
C09822=1203.863,-11.282,-42.561,-179.850,5.567,148.934
C09823=1203.858,-11.033,-42.574,-179.847,5.568,148.933
C09824=1203.853,-10.783,-42.588,-179.845,5.568,148.932
C09825=1203.848,-10.534,-42.600,-179.842,5.569,148.932
C09826=1203.843,-10.284,-42.615,-179.840,5.568,148.931
C09827=1203.837,-10.034,-42.628,-179.837,5.569,148.930
C09828=1203.833,-9.785,-42.642,-179.835,5.569,148.930
C09829=1203.827,-9.535,-42.655,-179.832,5.570,148.929
C09830=1203.822,-9.286,-42.669,-179.830,5.571,148.929
C09831=1203.818,-9.036,-42.683,-179.828,5.570,148.928
C09832=1203.812,-8.786,-42.696,-179.825,5.571,148.927
C09833=1203.807,-8.537,-42.710,-179.822,5.571,148.926
C09834=1203.802,-8.287,-42.723,-179.820,5.572,148.926
C09835=1203.797,-8.038,-42.737,-179.817,5.572,148.925
C09836=1203.792,-7.788,-42.751,-179.814,5.573,148.924
C09837=1203.787,-7.538,-42.764,-179.813,5.573,148.924
C09838=1203.782,-7.289,-42.778,-179.810,5.573,148.923
C09839=1203.776,-7.039,-42.792,-179.808,5.574,148.923
C09840=1203.772,-6.790,-42.805,-179.805,5.574,148.922
C09841=1203.767,-6.540,-42.819,-179.802,5.575,148.921
C09842=1203.761,-6.290,-42.833,-179.800,5.574,148.920
C09843=1203.756,-6.041,-42.847,-179.798,5.575,148.920
C09844=1203.752,-5.792,-42.861,-179.795,5.576,148.919
C09845=1203.747,-5.542,-42.875,-179.793,5.576,148.919
C09846=1203.741,-5.292,-42.888,-179.790,5.577,148.918
C09847=1203.736,-5.043,-42.902,-179.787,5.577,148.917
C09848=1203.731,-4.794,-42.916,-179.785,5.577,148.917
C09849=1203.726,-4.544,-42.929,-179.783,5.577,148.916
C09850=1203.721,-4.294,-42.944,-179.780,5.578,148.915
C09851=1203.715,-4.045,-42.957,-179.778,5.579,148.915
C09852=1203.711,-3.796,-42.971,-179.775,5.579,148.914
C09853=1203.706,-3.545,-42.985,-179.773,5.580,148.913
C09854=1203.700,-3.296,-42.999,-179.770,5.580,148.913
C09855=1203.695,-3.046,-43.013,-179.768,5.580,148.912
C09856=1203.690,-2.797,-43.027,-179.765,5.580,148.911
C09857=1203.685,-2.547,-43.040,-179.763,5.581,148.911
C09858=1203.680,-2.298,-43.054,-179.760,5.582,148.910
C09859=1203.675,-2.048,-43.068,-179.758,5.582,148.909
C09860=1203.670,-1.798,-43.083,-179.755,5.583,148.909
C09861=1203.665,-1.549,-43.096,-179.753,5.582,148.908
C09862=1203.660,-1.299,-43.109,-179.750,5.583,148.907
C09863=1203.655,-1.050,-43.124,-179.748,5.583,148.907
C09864=1203.650,-0.801,-43.138,-179.745,5.584,148.906
C09865=1203.645,-0.551,-43.152,-179.743,5.585,148.906
C09866=1203.640,-0.301,-43.166,-179.740,5.585,148.905
C09867=1203.634,-0.052,-43.180,-179.738,5.586,148.904
C09868=1203.629,0.198,-43.194,-179.735,5.585,148.903
C09869=1203.625,0.448,-43.207,-179.733,5.586,148.903
C09870=1203.620,0.697,-43.222,-179.730,5.586,148.902
C09871=1203.614,0.946,-43.236,-179.728,5.587,148.902
C09872=1203.609,1.196,-43.250,-179.725,5.588,148.901
C09873=1203.604,1.446,-43.264,-179.723,5.588,148.900
C09874=1203.599,1.695,-43.278,-179.720,5.589,148.900
C09875=1203.594,1.944,-43.292,-179.718,5.588,148.899
C09876=1203.589,2.194,-43.307,-179.715,5.589,148.898
C09877=1203.584,2.444,-43.321,-179.713,5.590,148.898
C09878=1203.578,2.713,-43.336,-179.710,5.590,148.897
C09879=1203.573,2.983,-43.351,-179.707,5.590,148.896
C09880=1203.567,3.251,-43.366,-179.705,5.591,148.895
C09881=1203.562,3.520,-43.381,-179.702,5.591,148.895
C09882=1203.557,3.770,-43.395,-179.699,5.592,148.894
C09883=1203.552,4.020,-43.410,-179.697,5.593,148.894
C09884=1203.547,4.269,-43.424,-179.695,5.593,148.893
C09885=1203.541,4.518,-43.438,-179.692,5.594,148.892
C09886=1203.536,4.768,-43.452,-179.689,5.594,148.892
C09887=1203.531,5.018,-43.466,-179.687,5.595,148.891
C09888=1203.527,5.268,-43.481,-179.685,5.594,148.890
C09889=1203.522,5.517,-43.495,-179.682,5.595,148.890
C09890=1203.516,5.766,-43.509,-179.680,5.596,148.889
C09891=1203.511,6.016,-43.523,-179.677,5.596,148.888
C09892=1203.506,6.266,-43.537,-179.674,5.597,148.888
C09893=1203.501,6.515,-43.552,-179.672,5.597,148.887
C09894=1203.497,6.764,-43.567,-179.669,5.598,148.886
C09895=1203.491,7.013,-43.581,-179.666,5.598,148.886
C09896=1203.486,7.263,-43.595,-179.665,5.598,148.885
C09897=1203.481,7.513,-43.609,-179.662,5.599,148.884
C09898=1203.476,7.763,-43.623,-179.660,5.599,148.884
C09899=1203.471,8.012,-43.638,-179.657,5.600,148.883
C09900=1203.466,8.262,-43.652,-179.654,5.600,148.882
C09901=1203.461,8.511,-43.666,-179.652,5.601,148.882
C09902=1203.456,8.760,-43.681,-179.649,5.602,148.881
C09903=1203.451,9.010,-43.695,-179.647,5.602,148.881
C09904=1203.446,9.260,-43.709,-179.644,5.603,148.880
C09905=1203.441,9.509,-43.724,-179.641,5.603,148.879
C09906=1203.436,9.759,-43.738,-179.639,5.603,148.878
C09907=1203.431,10.009,-43.752,-179.637,5.604,148.878
C09908=1203.426,10.257,-43.767,-179.635,5.604,148.877
C09909=1203.420,10.507,-43.782,-179.632,5.605,148.877
C09910=1203.415,10.757,-43.796,-179.629,5.605,148.876
C09911=1203.410,11.006,-43.810,-179.627,5.606,148.875
C09912=1203.405,11.256,-43.825,-179.624,5.606,148.875
C09913=1203.401,11.505,-43.840,-179.621,5.607,148.874
C09914=1203.396,11.755,-43.854,-179.619,5.608,148.873
C09915=1203.391,12.005,-43.868,-179.617,5.608,148.873
C09916=1203.385,12.255,-43.883,-179.614,5.609,148.872
C09917=1203.381,12.504,-43.898,-179.612,5.609,148.871
C09918=1203.375,12.753,-43.912,-179.609,5.609,148.871
C09919=1203.370,13.003,-43.926,-179.607,5.610,148.870
C09920=1203.365,13.252,-43.941,-179.604,5.610,148.870
C09921=1203.360,13.501,-43.956,-179.602,5.611,148.869
C09922=1203.355,13.751,-43.970,-179.599,5.611,148.868
C09923=1203.350,14.001,-43.985,-179.596,5.612,148.868
C09924=1203.345,14.250,-44.000,-179.594,5.612,148.867
C09925=1203.340,14.500,-44.014,-179.592,5.613,148.866
C09926=1203.335,14.750,-44.028,-179.589,5.614,148.866
C09927=1203.331,14.999,-44.043,-179.586,5.614,148.865
C09928=1203.325,15.249,-44.058,-179.584,5.615,148.864
C09929=1203.320,15.498,-44.073,-179.582,5.615,148.864
C09930=1203.315,15.748,-44.087,-179.579,5.615,148.863
C09931=1203.310,15.997,-44.102,-179.577,5.616,148.863
C09932=1203.305,16.247,-44.117,-179.574,5.616,148.862
C09933=1203.300,16.496,-44.131,-179.571,5.617,148.861
C09934=1203.295,16.745,-44.146,-179.569,5.617,148.860
C09935=1203.290,16.994,-44.160,-179.566,5.618,148.860
C09936=1203.284,17.244,-44.175,-179.564,5.618,148.859
C09937=1203.279,17.494,-44.190,-179.561,5.619,148.859
C09938=1203.274,17.743,-44.205,-179.559,5.620,148.858
C09939=1203.270,17.992,-44.220,-179.556,5.620,148.857
C09940=1203.264,18.242,-44.234,-179.553,5.621,148.857
C09941=1203.259,18.491,-44.249,-179.551,5.621,148.856
C09942=1203.254,18.741,-44.264,-179.549,5.622,148.855
C09943=1203.249,18.991,-44.279,-179.546,5.623,148.855
C09944=1203.244,19.240,-44.294,-179.543,5.623,148.854
C09945=1203.240,19.489,-44.309,-179.541,5.623,148.853
C09946=1203.235,19.739,-44.323,-179.539,5.624,148.853
C09947=1203.230,19.989,-44.339,-179.536,5.624,148.852
C09948=1203.225,20.239,-44.353,-179.534,5.625,148.852
C09949=1203.220,20.488,-44.368,-179.531,5.625,148.851
C09950=1203.214,20.738,-44.383,-179.529,5.626,148.850
C09951=1203.210,20.987,-44.398,-179.526,5.626,148.850
C09952=1203.204,21.237,-44.413,-179.523,5.627,148.849
C09953=1203.199,21.486,-44.428,-179.521,5.628,148.848
C09954=1203.195,21.736,-44.442,-179.518,5.628,148.848
C09955=1203.189,21.985,-44.458,-179.516,5.629,148.847
C09956=1203.184,22.234,-44.473,-179.513,5.629,148.846
C09957=1203.180,22.484,-44.487,-179.510,5.630,148.846
C09958=1203.174,22.734,-44.502,-179.508,5.631,148.845
C09959=1203.169,22.983,-44.517,-179.506,5.631,148.845
C09960=1203.164,23.233,-44.532,-179.503,5.632,148.844
C09961=1203.159,23.482,-44.547,-179.500,5.632,148.843
C09962=1203.154,23.731,-44.562,-179.498,5.633,148.843
C09963=1203.149,23.981,-44.577,-179.496,5.634,148.842
C09964=1203.144,24.230,-44.592,-179.493,5.634,148.841
C09965=1203.139,24.481,-44.607,-179.490,5.635,148.841
C09966=1203.134,24.730,-44.622,-179.488,5.635,148.840
C09967=1203.130,24.979,-44.637,-179.485,5.636,148.839
C09968=1203.124,25.229,-44.652,-179.483,5.637,148.839
C09969=1203.119,25.478,-44.667,-179.480,5.637,148.838
C09970=1203.114,25.727,-44.683,-179.478,5.637,148.838
C09971=1203.109,25.977,-44.697,-179.475,5.637,148.837
C09972=1203.104,26.226,-44.713,-179.473,5.638,148.836
C09973=1203.099,26.476,-44.728,-179.471,5.639,148.836
C09974=1203.094,26.726,-44.744,-179.468,5.639,148.835
C09975=1203.089,26.975,-44.758,-179.465,5.640,148.834
C09976=1203.084,27.225,-44.774,-179.463,5.640,148.834
C09977=1203.079,27.474,-44.789,-179.460,5.641,148.833
C09978=1203.074,27.723,-44.804,-179.458,5.642,148.833
C09979=1203.069,27.973,-44.818,-179.455,5.642,148.832
C09980=1203.064,28.222,-44.834,-179.453,5.643,148.831
C09981=1203.059,28.472,-44.849,-179.450,5.643,148.831
C09982=1203.054,28.741,-44.866,-179.447,5.644,148.830
C09983=1203.049,29.009,-44.882,-179.444,5.645,148.829
C09984=1203.043,29.279,-44.898,-179.441,5.646,148.829
C09985=1203.037,29.547,-44.915,-179.439,5.646,148.828
C09986=1203.033,29.796,-44.930,-179.436,5.647,148.827
C09987=1203.027,30.046,-44.945,-179.434,5.648,148.827
C09988=1203.022,30.295,-44.960,-179.431,5.648,148.826
C09989=1203.017,30.545,-44.976,-179.429,5.649,148.825
C09990=1203.013,30.794,-44.991,-179.426,5.649,148.825
C09991=1203.008,31.044,-45.007,-179.423,5.650,148.824
C09992=1203.002,31.293,-45.022,-179.421,5.651,148.824
C09993=1202.998,31.542,-45.037,-179.419,5.651,148.823
C09994=1202.992,31.792,-45.053,-179.416,5.652,148.822
C09995=1202.988,32.042,-45.068,-179.413,5.652,148.822
C09996=1202.982,32.292,-45.083,-179.411,5.653,148.821
//INST
///DATE 2021/06/15 17:23
///ATTR SC,RW,RJ
////FRAME ROBOT
///GROUP1 RB1
NOP
MOVL C00000 V=800.0 PL=0
MOVL C00001 V=800.0 PL=0
MOVL C00002 V=800.0 PL=0
MOVL C00003 V=800.0 PL=0
MOVL C00004 V=800.0 PL=0
MOVL C00005 V=800.0 PL=0
MOVL C00006 V=800.0 PL=0
MOVL C00007 V=800.0 PL=0
MOVL C00008 V=800.0 PL=0
MOVL C00009 V=800.0 PL=0
MOVL C00010 V=800.0 PL=0
MOVL C00011 V=800.0 PL=0
MOVL C00012 V=800.0 PL=0
MOVL C00013 V=800.0 PL=0
MOVL C00014 V=800.0 PL=0
MOVL C00015 V=800.0 PL=0
MOVL C00016 V=800.0 PL=0
MOVL C00017 V=800.0 PL=0
MOVL C00018 V=800.0 PL=0
MOVL C00019 V=800.0 PL=0
MOVL C00020 V=800.0 PL=0
MOVL C00021 V=800.0 PL=0
MOVL C00022 V=800.0 PL=0
MOVL C00023 V=800.0 PL=0
MOVL C00024 V=800.0 PL=0
MOVL C00025 V=800.0 PL=0
MOVL C00026 V=800.0 PL=0
MOVL C00027 V=800.0 PL=0
MOVL C00028 V=800.0 PL=0
MOVL C00029 V=800.0 PL=0
MOVL C00030 V=800.0 PL=0
MOVL C00031 V=800.0 PL=0
MOVL C00032 V=800.0 PL=0
MOVL C00033 V=800.0 PL=0
MOVL C00034 V=800.0 PL=0
MOVL C00035 V=800.0 PL=0
MOVL C00036 V=800.0 PL=0
MOVL C00037 V=800.0 PL=0
MOVL C00038 V=800.0 PL=0
MOVL C00039 V=800.0 PL=0
MOVL C00040 V=800.0 PL=0
MOVL C00041 V=800.0 PL=0
MOVL C00042 V=800.0 PL=0
MOVL C00043 V=800.0 PL=0
MOVL C00044 V=800.0 PL=0
MOVL C00045 V=800.0 PL=0
MOVL C00046 V=800.0 PL=0
MOVL C00047 V=800.0 PL=0
MOVL C00048 V=800.0 PL=0
MOVL C00049 V=800.0 PL=0
MOVL C00050 V=800.0 PL=0
MOVL C00051 V=800.0 PL=0
MOVL C00052 V=800.0 PL=0
MOVL C00053 V=800.0 PL=0
MOVL C00054 V=800.0 PL=0
MOVL C00055 V=800.0 PL=0
MOVL C00056 V=800.0 PL=0
MOVL C00057 V=800.0 PL=0
MOVL C00058 V=800.0 PL=0
MOVL C00059 V=800.0 PL=0
MOVL C00060 V=800.0 PL=0
MOVL C00061 V=800.0 PL=0
MOVL C00062 V=800.0 PL=0
MOVL C00063 V=800.0 PL=0
MOVL C00064 V=800.0 PL=0
MOVL C00065 V=800.0 PL=0
MOVL C00066 V=800.0 PL=0
MOVL C00067 V=800.0 PL=0
MOVL C00068 V=800.0 PL=0
MOVL C00069 V=800.0 PL=0
MOVL C00070 V=800.0 PL=0
MOVL C00071 V=800.0 PL=0
MOVL C00072 V=800.0 PL=0
MOVL C00073 V=800.0 PL=0
MOVL C00074 V=800.0 PL=0
MOVL C00075 V=800.0 PL=0
MOVL C00076 V=800.0 PL=0
MOVL C00077 V=800.0 PL=0
MOVL C00078 V=800.0 PL=0
MOVL C00079 V=800.0 PL=0
MOVL C00080 V=800.0 PL=0
MOVL C00081 V=800.0 PL=0
MOVL C00082 V=800.0 PL=0
MOVL C00083 V=800.0 PL=0
MOVL C00084 V=800.0 PL=0
MOVL C00085 V=800.0 PL=0
MOVL C00086 V=800.0 PL=0
MOVL C00087 V=800.0 PL=0
MOVL C00088 V=800.0 PL=0
MOVL C00089 V=800.0 PL=0
MOVL C00090 V=800.0 PL=0
MOVL C00091 V=800.0 PL=0
MOVL C00092 V=800.0 PL=0
MOVL C00093 V=800.0 PL=0
MOVL C00094 V=800.0 PL=0
MOVL C00095 V=800.0 PL=0
MOVL C00096 V=800.0 PL=0
MOVL C00097 V=800.0 PL=0
MOVL C00098 V=800.0 PL=0
MOVL C00099 V=800.0 PL=0
MOVL C00100 V=800.0 PL=0
MOVL C00101 V=800.0 PL=0
MOVL C00102 V=800.0 PL=0
MOVL C00103 V=800.0 PL=0
MOVL C00104 V=800.0 PL=0
MOVL C00105 V=800.0 PL=0
MOVL C00106 V=800.0 PL=0
MOVL C00107 V=800.0 PL=0
MOVL C00108 V=800.0 PL=0
MOVL C00109 V=800.0 PL=0
MOVL C00110 V=800.0 PL=0
MOVL C00111 V=800.0 PL=0
MOVL C00112 V=800.0 PL=0
MOVL C00113 V=800.0 PL=0
MOVL C00114 V=800.0 PL=0
MOVL C00115 V=800.0 PL=0
MOVL C00116 V=800.0 PL=0
MOVL C00117 V=800.0 PL=0
MOVL C00118 V=800.0 PL=0
MOVL C00119 V=800.0 PL=0
MOVL C00120 V=800.0 PL=0
MOVL C00121 V=800.0 PL=0
MOVL C00122 V=800.0 PL=0
MOVL C00123 V=800.0 PL=0
MOVL C00124 V=800.0 PL=0
MOVL C00125 V=800.0 PL=0
MOVL C00126 V=800.0 PL=0
MOVL C00127 V=800.0 PL=0
MOVL C00128 V=800.0 PL=0
MOVL C00129 V=800.0 PL=0
MOVL C00130 V=800.0 PL=0
MOVL C00131 V=800.0 PL=0
MOVL C00132 V=800.0 PL=0
MOVL C00133 V=800.0 PL=0
MOVL C00134 V=800.0 PL=0
MOVL C00135 V=800.0 PL=0
MOVL C00136 V=800.0 PL=0
MOVL C00137 V=800.0 PL=0
MOVL C00138 V=800.0 PL=0
MOVL C00139 V=800.0 PL=0
MOVL C00140 V=800.0 PL=0
MOVL C00141 V=800.0 PL=0
MOVL C00142 V=800.0 PL=0
MOVL C00143 V=800.0 PL=0
MOVL C00144 V=800.0 PL=0
MOVL C00145 V=800.0 PL=0
MOVL C00146 V=800.0 PL=0
MOVL C00147 V=800.0 PL=0
MOVL C00148 V=800.0 PL=0
MOVL C00149 V=800.0 PL=0
MOVL C00150 V=800.0 PL=0
MOVL C00151 V=800.0 PL=0
MOVL C00152 V=800.0 PL=0
MOVL C00153 V=800.0 PL=0
MOVL C00154 V=800.0 PL=0
MOVL C00155 V=800.0 PL=0
MOVL C00156 V=800.0 PL=0
MOVL C00157 V=800.0 PL=0
MOVL C00158 V=800.0 PL=0
MOVL C00159 V=800.0 PL=0
MOVL C00160 V=800.0 PL=0
MOVL C00161 V=800.0 PL=0
MOVL C00162 V=800.0 PL=0
MOVL C00163 V=800.0 PL=0
MOVL C00164 V=800.0 PL=0
MOVL C00165 V=800.0 PL=0
MOVL C00166 V=800.0 PL=0
MOVL C00167 V=800.0 PL=0
MOVL C00168 V=800.0 PL=0
MOVL C00169 V=800.0 PL=0
MOVL C00170 V=800.0 PL=0
MOVL C00171 V=800.0 PL=0
MOVL C00172 V=800.0 PL=0
MOVL C00173 V=800.0 PL=0
MOVL C00174 V=800.0 PL=0
MOVL C00175 V=800.0 PL=0
MOVL C00176 V=800.0 PL=0
MOVL C00177 V=800.0 PL=0
MOVL C00178 V=800.0 PL=0
MOVL C00179 V=800.0 PL=0
MOVL C00180 V=800.0 PL=0
MOVL C00181 V=800.0 PL=0
MOVL C00182 V=800.0 PL=0
MOVL C00183 V=800.0 PL=0
MOVL C00184 V=800.0 PL=0
MOVL C00185 V=800.0 PL=0
MOVL C00186 V=800.0 PL=0
MOVL C00187 V=800.0 PL=0
MOVL C00188 V=800.0 PL=0
MOVL C00189 V=800.0 PL=0
MOVL C00190 V=800.0 PL=0
MOVL C00191 V=800.0 PL=0
MOVL C00192 V=800.0 PL=0
MOVL C00193 V=800.0 PL=0
MOVL C00194 V=800.0 PL=0
MOVL C00195 V=800.0 PL=0
MOVL C00196 V=800.0 PL=0
MOVL C00197 V=800.0 PL=0
MOVL C00198 V=800.0 PL=0
MOVL C00199 V=800.0 PL=0
MOVL C00200 V=800.0 PL=0
MOVL C00201 V=800.0 PL=0
MOVL C00202 V=800.0 PL=0
MOVL C00203 V=800.0 PL=0
MOVL C00204 V=800.0 PL=0
MOVL C00205 V=800.0 PL=0
MOVL C00206 V=800.0 PL=0
MOVL C00207 V=800.0 PL=0
MOVL C00208 V=800.0 PL=0
MOVL C00209 V=800.0 PL=0
MOVL C00210 V=800.0 PL=0
MOVL C00211 V=800.0 PL=0
MOVL C00212 V=800.0 PL=0
MOVL C00213 V=800.0 PL=0
MOVL C00214 V=800.0 PL=0
MOVL C00215 V=800.0 PL=0
MOVL C00216 V=800.0 PL=0
MOVL C00217 V=800.0 PL=0
MOVL C00218 V=800.0 PL=0
MOVL C00219 V=800.0 PL=0
MOVL C00220 V=800.0 PL=0
MOVL C00221 V=800.0 PL=0
MOVL C00222 V=800.0 PL=0
MOVL C00223 V=800.0 PL=0
MOVL C00224 V=800.0 PL=0
MOVL C00225 V=800.0 PL=0
MOVL C00226 V=800.0 PL=0
MOVL C00227 V=800.0 PL=0
MOVL C00228 V=800.0 PL=0
MOVL C00229 V=800.0 PL=0
MOVL C00230 V=800.0 PL=0
MOVL C00231 V=800.0 PL=0
MOVL C00232 V=800.0 PL=0
MOVL C00233 V=800.0 PL=0
MOVL C00234 V=800.0 PL=0
MOVL C00235 V=800.0 PL=0
MOVL C00236 V=800.0 PL=0
MOVL C00237 V=800.0 PL=0
MOVL C00238 V=800.0 PL=0
MOVL C00239 V=800.0 PL=0
MOVL C00240 V=800.0 PL=0
MOVL C00241 V=800.0 PL=0
MOVL C00242 V=800.0 PL=0
MOVL C00243 V=800.0 PL=0
MOVL C00244 V=800.0 PL=0
MOVL C00245 V=800.0 PL=0
MOVL C00246 V=800.0 PL=0
MOVL C00247 V=800.0 PL=0
MOVL C00248 V=800.0 PL=0
MOVL C00249 V=800.0 PL=0
MOVL C00250 V=800.0 PL=0
MOVL C00251 V=800.0 PL=0
MOVL C00252 V=800.0 PL=0
MOVL C00253 V=800.0 PL=0
MOVL C00254 V=800.0 PL=0
MOVL C00255 V=800.0 PL=0
MOVL C00256 V=800.0 PL=0
MOVL C00257 V=800.0 PL=0
MOVL C00258 V=800.0 PL=0
MOVL C00259 V=800.0 PL=0
MOVL C00260 V=800.0 PL=0
MOVL C00261 V=800.0 PL=0
MOVL C00262 V=800.0 PL=0
MOVL C00263 V=800.0 PL=0
MOVL C00264 V=800.0 PL=0
MOVL C00265 V=800.0 PL=0
MOVL C00266 V=800.0 PL=0
MOVL C00267 V=800.0 PL=0
MOVL C00268 V=800.0 PL=0
MOVL C00269 V=800.0 PL=0
MOVL C00270 V=800.0 PL=0
MOVL C00271 V=800.0 PL=0
MOVL C00272 V=800.0 PL=0
MOVL C00273 V=800.0 PL=0
MOVL C00274 V=800.0 PL=0
MOVL C00275 V=800.0 PL=0
MOVL C00276 V=800.0 PL=0
MOVL C00277 V=800.0 PL=0
MOVL C00278 V=800.0 PL=0
MOVL C00279 V=800.0 PL=0
MOVL C00280 V=800.0 PL=0
MOVL C00281 V=800.0 PL=0
MOVL C00282 V=800.0 PL=0
MOVL C00283 V=800.0 PL=0
MOVL C00284 V=800.0 PL=0
MOVL C00285 V=800.0 PL=0
MOVL C00286 V=800.0 PL=0
MOVL C00287 V=800.0 PL=0
MOVL C00288 V=800.0 PL=0
MOVL C00289 V=800.0 PL=0
MOVL C00290 V=800.0 PL=0
MOVL C00291 V=800.0 PL=0
MOVL C00292 V=800.0 PL=0
MOVL C00293 V=800.0 PL=0
MOVL C00294 V=800.0 PL=0
MOVL C00295 V=800.0 PL=0
MOVL C00296 V=800.0 PL=0
MOVL C00297 V=800.0 PL=0
MOVL C00298 V=800.0 PL=0
MOVL C00299 V=800.0 PL=0
MOVL C00300 V=800.0 PL=0
MOVL C00301 V=800.0 PL=0
MOVL C00302 V=800.0 PL=0
MOVL C00303 V=800.0 PL=0
MOVL C00304 V=800.0 PL=0
MOVL C00305 V=800.0 PL=0
MOVL C00306 V=800.0 PL=0
MOVL C00307 V=800.0 PL=0
MOVL C00308 V=800.0 PL=0
MOVL C00309 V=800.0 PL=0
MOVL C00310 V=800.0 PL=0
MOVL C00311 V=800.0 PL=0
MOVL C00312 V=800.0 PL=0
MOVL C00313 V=800.0 PL=0
MOVL C00314 V=800.0 PL=0
MOVL C00315 V=800.0 PL=0
MOVL C00316 V=800.0 PL=0
MOVL C00317 V=800.0 PL=0
MOVL C00318 V=800.0 PL=0
MOVL C00319 V=800.0 PL=0
MOVL C00320 V=800.0 PL=0
MOVL C00321 V=800.0 PL=0
MOVL C00322 V=800.0 PL=0
MOVL C00323 V=800.0 PL=0
MOVL C00324 V=800.0 PL=0
MOVL C00325 V=800.0 PL=0
MOVL C00326 V=800.0 PL=0
MOVL C00327 V=800.0 PL=0
MOVL C00328 V=800.0 PL=0
MOVL C00329 V=800.0 PL=0
MOVL C00330 V=800.0 PL=0
MOVL C00331 V=800.0 PL=0
MOVL C00332 V=800.0 PL=0
MOVL C00333 V=800.0 PL=0
MOVL C00334 V=800.0 PL=0
MOVL C00335 V=800.0 PL=0
MOVL C00336 V=800.0 PL=0
MOVL C00337 V=800.0 PL=0
MOVL C00338 V=800.0 PL=0
MOVL C00339 V=800.0 PL=0
MOVL C00340 V=800.0 PL=0
MOVL C00341 V=800.0 PL=0
MOVL C00342 V=800.0 PL=0
MOVL C00343 V=800.0 PL=0
MOVL C00344 V=800.0 PL=0
MOVL C00345 V=800.0 PL=0
MOVL C00346 V=800.0 PL=0
MOVL C00347 V=800.0 PL=0
MOVL C00348 V=800.0 PL=0
MOVL C00349 V=800.0 PL=0
MOVL C00350 V=800.0 PL=0
MOVL C00351 V=800.0 PL=0
MOVL C00352 V=800.0 PL=0
MOVL C00353 V=800.0 PL=0
MOVL C00354 V=800.0 PL=0
MOVL C00355 V=800.0 PL=0
MOVL C00356 V=800.0 PL=0
MOVL C00357 V=800.0 PL=0
MOVL C00358 V=800.0 PL=0
MOVL C00359 V=800.0 PL=0
MOVL C00360 V=800.0 PL=0
MOVL C00361 V=800.0 PL=0
MOVL C00362 V=800.0 PL=0
MOVL C00363 V=800.0 PL=0
MOVL C00364 V=800.0 PL=0
MOVL C00365 V=800.0 PL=0
MOVL C00366 V=800.0 PL=0
MOVL C00367 V=800.0 PL=0
MOVL C00368 V=800.0 PL=0
MOVL C00369 V=800.0 PL=0
MOVL C00370 V=800.0 PL=0
MOVL C00371 V=800.0 PL=0
MOVL C00372 V=800.0 PL=0
MOVL C00373 V=800.0 PL=0
MOVL C00374 V=800.0 PL=0
MOVL C00375 V=800.0 PL=0
MOVL C00376 V=800.0 PL=0
MOVL C00377 V=800.0 PL=0
MOVL C00378 V=800.0 PL=0
MOVL C00379 V=800.0 PL=0
MOVL C00380 V=800.0 PL=0
MOVL C00381 V=800.0 PL=0
MOVL C00382 V=800.0 PL=0
MOVL C00383 V=800.0 PL=0
MOVL C00384 V=800.0 PL=0
MOVL C00385 V=800.0 PL=0
MOVL C00386 V=800.0 PL=0
MOVL C00387 V=800.0 PL=0
MOVL C00388 V=800.0 PL=0
MOVL C00389 V=800.0 PL=0
MOVL C00390 V=800.0 PL=0
MOVL C00391 V=800.0 PL=0
MOVL C00392 V=800.0 PL=0
MOVL C00393 V=800.0 PL=0
MOVL C00394 V=800.0 PL=0
MOVL C00395 V=800.0 PL=0
MOVL C00396 V=800.0 PL=0
MOVL C00397 V=800.0 PL=0
MOVL C00398 V=800.0 PL=0
MOVL C00399 V=800.0 PL=0
MOVL C00400 V=800.0 PL=0
MOVL C00401 V=800.0 PL=0
MOVL C00402 V=800.0 PL=0
MOVL C00403 V=800.0 PL=0
MOVL C00404 V=800.0 PL=0
MOVL C00405 V=800.0 PL=0
MOVL C00406 V=800.0 PL=0
MOVL C00407 V=800.0 PL=0
MOVL C00408 V=800.0 PL=0
MOVL C00409 V=800.0 PL=0
MOVL C00410 V=800.0 PL=0
MOVL C00411 V=800.0 PL=0
MOVL C00412 V=800.0 PL=0
MOVL C00413 V=800.0 PL=0
MOVL C00414 V=800.0 PL=0
MOVL C00415 V=800.0 PL=0
MOVL C00416 V=800.0 PL=0
MOVL C00417 V=800.0 PL=0
MOVL C00418 V=800.0 PL=0
MOVL C00419 V=800.0 PL=0
MOVL C00420 V=800.0 PL=0
MOVL C00421 V=800.0 PL=0
MOVL C00422 V=800.0 PL=0
MOVL C00423 V=800.0 PL=0
MOVL C00424 V=800.0 PL=0
MOVL C00425 V=800.0 PL=0
MOVL C00426 V=800.0 PL=0
MOVL C00427 V=800.0 PL=0
MOVL C00428 V=800.0 PL=0
MOVL C00429 V=800.0 PL=0
MOVL C00430 V=800.0 PL=0
MOVL C00431 V=800.0 PL=0
MOVL C00432 V=800.0 PL=0
MOVL C00433 V=800.0 PL=0
MOVL C00434 V=800.0 PL=0
MOVL C00435 V=800.0 PL=0
MOVL C00436 V=800.0 PL=0
MOVL C00437 V=800.0 PL=0
MOVL C00438 V=800.0 PL=0
MOVL C00439 V=800.0 PL=0
MOVL C00440 V=800.0 PL=0
MOVL C00441 V=800.0 PL=0
MOVL C00442 V=800.0 PL=0
MOVL C00443 V=800.0 PL=0
MOVL C00444 V=800.0 PL=0
MOVL C00445 V=800.0 PL=0
MOVL C00446 V=800.0 PL=0
MOVL C00447 V=800.0 PL=0
MOVL C00448 V=800.0 PL=0
MOVL C00449 V=800.0 PL=0
MOVL C00450 V=800.0 PL=0
MOVL C00451 V=800.0 PL=0
MOVL C00452 V=800.0 PL=0
MOVL C00453 V=800.0 PL=0
MOVL C00454 V=800.0 PL=0
MOVL C00455 V=800.0 PL=0
MOVL C00456 V=800.0 PL=0
MOVL C00457 V=800.0 PL=0
MOVL C00458 V=800.0 PL=0
MOVL C00459 V=800.0 PL=0
MOVL C00460 V=800.0 PL=0
MOVL C00461 V=800.0 PL=0
MOVL C00462 V=800.0 PL=0
MOVL C00463 V=800.0 PL=0
MOVL C00464 V=800.0 PL=0
MOVL C00465 V=800.0 PL=0
MOVL C00466 V=800.0 PL=0
MOVL C00467 V=800.0 PL=0
MOVL C00468 V=800.0 PL=0
MOVL C00469 V=800.0 PL=0
MOVL C00470 V=800.0 PL=0
MOVL C00471 V=800.0 PL=0
MOVL C00472 V=800.0 PL=0
MOVL C00473 V=800.0 PL=0
MOVL C00474 V=800.0 PL=0
MOVL C00475 V=800.0 PL=0
MOVL C00476 V=800.0 PL=0
MOVL C00477 V=800.0 PL=0
MOVL C00478 V=800.0 PL=0
MOVL C00479 V=800.0 PL=0
MOVL C00480 V=800.0 PL=0
MOVL C00481 V=800.0 PL=0
MOVL C00482 V=800.0 PL=0
MOVL C00483 V=800.0 PL=0
MOVL C00484 V=800.0 PL=0
MOVL C00485 V=800.0 PL=0
MOVL C00486 V=800.0 PL=0
MOVL C00487 V=800.0 PL=0
MOVL C00488 V=800.0 PL=0
MOVL C00489 V=800.0 PL=0
MOVL C00490 V=800.0 PL=0
MOVL C00491 V=800.0 PL=0
MOVL C00492 V=800.0 PL=0
MOVL C00493 V=800.0 PL=0
MOVL C00494 V=800.0 PL=0
MOVL C00495 V=800.0 PL=0
MOVL C00496 V=800.0 PL=0
MOVL C00497 V=800.0 PL=0
MOVL C00498 V=800.0 PL=0
MOVL C00499 V=800.0 PL=0
MOVL C00500 V=800.0 PL=0
MOVL C00501 V=800.0 PL=0
MOVL C00502 V=800.0 PL=0
MOVL C00503 V=800.0 PL=0
MOVL C00504 V=800.0 PL=0
MOVL C00505 V=800.0 PL=0
MOVL C00506 V=800.0 PL=0
MOVL C00507 V=800.0 PL=0
MOVL C00508 V=800.0 PL=0
MOVL C00509 V=800.0 PL=0
MOVL C00510 V=800.0 PL=0
MOVL C00511 V=800.0 PL=0
MOVL C00512 V=800.0 PL=0
MOVL C00513 V=800.0 PL=0
MOVL C00514 V=800.0 PL=0
MOVL C00515 V=800.0 PL=0
MOVL C00516 V=800.0 PL=0
MOVL C00517 V=800.0 PL=0
MOVL C00518 V=800.0 PL=0
MOVL C00519 V=800.0 PL=0
MOVL C00520 V=800.0 PL=0
MOVL C00521 V=800.0 PL=0
MOVL C00522 V=800.0 PL=0
MOVL C00523 V=800.0 PL=0
MOVL C00524 V=800.0 PL=0
MOVL C00525 V=800.0 PL=0
MOVL C00526 V=800.0 PL=0
MOVL C00527 V=800.0 PL=0
MOVL C00528 V=800.0 PL=0
MOVL C00529 V=800.0 PL=0
MOVL C00530 V=800.0 PL=0
MOVL C00531 V=800.0 PL=0
MOVL C00532 V=800.0 PL=0
MOVL C00533 V=800.0 PL=0
MOVL C00534 V=800.0 PL=0
MOVL C00535 V=800.0 PL=0
MOVL C00536 V=800.0 PL=0
MOVL C00537 V=800.0 PL=0
MOVL C00538 V=800.0 PL=0
MOVL C00539 V=800.0 PL=0
MOVL C00540 V=800.0 PL=0
MOVL C00541 V=800.0 PL=0
MOVL C00542 V=800.0 PL=0
MOVL C00543 V=800.0 PL=0
MOVL C00544 V=800.0 PL=0
MOVL C00545 V=800.0 PL=0
MOVL C00546 V=800.0 PL=0
MOVL C00547 V=800.0 PL=0
MOVL C00548 V=800.0 PL=0
MOVL C00549 V=800.0 PL=0
MOVL C00550 V=800.0 PL=0
MOVL C00551 V=800.0 PL=0
MOVL C00552 V=800.0 PL=0
MOVL C00553 V=800.0 PL=0
MOVL C00554 V=800.0 PL=0
MOVL C00555 V=800.0 PL=0
MOVL C00556 V=800.0 PL=0
MOVL C00557 V=800.0 PL=0
MOVL C00558 V=800.0 PL=0
MOVL C00559 V=800.0 PL=0
MOVL C00560 V=800.0 PL=0
MOVL C00561 V=800.0 PL=0
MOVL C00562 V=800.0 PL=0
MOVL C00563 V=800.0 PL=0
MOVL C00564 V=800.0 PL=0
MOVL C00565 V=800.0 PL=0
MOVL C00566 V=800.0 PL=0
MOVL C00567 V=800.0 PL=0
MOVL C00568 V=800.0 PL=0
MOVL C00569 V=800.0 PL=0
MOVL C00570 V=800.0 PL=0
MOVL C00571 V=800.0 PL=0
MOVL C00572 V=800.0 PL=0
MOVL C00573 V=800.0 PL=0
MOVL C00574 V=800.0 PL=0
MOVL C00575 V=800.0 PL=0
MOVL C00576 V=800.0 PL=0
MOVL C00577 V=800.0 PL=0
MOVL C00578 V=800.0 PL=0
MOVL C00579 V=800.0 PL=0
MOVL C00580 V=800.0 PL=0
MOVL C00581 V=800.0 PL=0
MOVL C00582 V=800.0 PL=0
MOVL C00583 V=800.0 PL=0
MOVL C00584 V=800.0 PL=0
MOVL C00585 V=800.0 PL=0
MOVL C00586 V=800.0 PL=0
MOVL C00587 V=800.0 PL=0
MOVL C00588 V=800.0 PL=0
MOVL C00589 V=800.0 PL=0
MOVL C00590 V=800.0 PL=0
MOVL C00591 V=800.0 PL=0
MOVL C00592 V=800.0 PL=0
MOVL C00593 V=800.0 PL=0
MOVL C00594 V=800.0 PL=0
MOVL C00595 V=800.0 PL=0
MOVL C00596 V=800.0 PL=0
MOVL C00597 V=800.0 PL=0
MOVL C00598 V=800.0 PL=0
MOVL C00599 V=800.0 PL=0
MOVL C00600 V=800.0 PL=0
MOVL C00601 V=800.0 PL=0
MOVL C00602 V=800.0 PL=0
MOVL C00603 V=800.0 PL=0
MOVL C00604 V=800.0 PL=0
MOVL C00605 V=800.0 PL=0
MOVL C00606 V=800.0 PL=0
MOVL C00607 V=800.0 PL=0
MOVL C00608 V=800.0 PL=0
MOVL C00609 V=800.0 PL=0
MOVL C00610 V=800.0 PL=0
MOVL C00611 V=800.0 PL=0
MOVL C00612 V=800.0 PL=0
MOVL C00613 V=800.0 PL=0
MOVL C00614 V=800.0 PL=0
MOVL C00615 V=800.0 PL=0
MOVL C00616 V=800.0 PL=0
MOVL C00617 V=800.0 PL=0
MOVL C00618 V=800.0 PL=0
MOVL C00619 V=800.0 PL=0
MOVL C00620 V=800.0 PL=0
MOVL C00621 V=800.0 PL=0
MOVL C00622 V=800.0 PL=0
MOVL C00623 V=800.0 PL=0
MOVL C00624 V=800.0 PL=0
MOVL C00625 V=800.0 PL=0
MOVL C00626 V=800.0 PL=0
MOVL C00627 V=800.0 PL=0
MOVL C00628 V=800.0 PL=0
MOVL C00629 V=800.0 PL=0
MOVL C00630 V=800.0 PL=0
MOVL C00631 V=800.0 PL=0
MOVL C00632 V=800.0 PL=0
MOVL C00633 V=800.0 PL=0
MOVL C00634 V=800.0 PL=0
MOVL C00635 V=800.0 PL=0
MOVL C00636 V=800.0 PL=0
MOVL C00637 V=800.0 PL=0
MOVL C00638 V=800.0 PL=0
MOVL C00639 V=800.0 PL=0
MOVL C00640 V=800.0 PL=0
MOVL C00641 V=800.0 PL=0
MOVL C00642 V=800.0 PL=0
MOVL C00643 V=800.0 PL=0
MOVL C00644 V=800.0 PL=0
MOVL C00645 V=800.0 PL=0
MOVL C00646 V=800.0 PL=0
MOVL C00647 V=800.0 PL=0
MOVL C00648 V=800.0 PL=0
MOVL C00649 V=800.0 PL=0
MOVL C00650 V=800.0 PL=0
MOVL C00651 V=800.0 PL=0
MOVL C00652 V=800.0 PL=0
MOVL C00653 V=800.0 PL=0
MOVL C00654 V=800.0 PL=0
MOVL C00655 V=800.0 PL=0
MOVL C00656 V=800.0 PL=0
MOVL C00657 V=800.0 PL=0
MOVL C00658 V=800.0 PL=0
MOVL C00659 V=800.0 PL=0
MOVL C00660 V=800.0 PL=0
MOVL C00661 V=800.0 PL=0
MOVL C00662 V=800.0 PL=0
MOVL C00663 V=800.0 PL=0
MOVL C00664 V=800.0 PL=0
MOVL C00665 V=800.0 PL=0
MOVL C00666 V=800.0 PL=0
MOVL C00667 V=800.0 PL=0
MOVL C00668 V=800.0 PL=0
MOVL C00669 V=800.0 PL=0
MOVL C00670 V=800.0 PL=0
MOVL C00671 V=800.0 PL=0
MOVL C00672 V=800.0 PL=0
MOVL C00673 V=800.0 PL=0
MOVL C00674 V=800.0 PL=0
MOVL C00675 V=800.0 PL=0
MOVL C00676 V=800.0 PL=0
MOVL C00677 V=800.0 PL=0
MOVL C00678 V=800.0 PL=0
MOVL C00679 V=800.0 PL=0
MOVL C00680 V=800.0 PL=0
MOVL C00681 V=800.0 PL=0
MOVL C00682 V=800.0 PL=0
MOVL C00683 V=800.0 PL=0
MOVL C00684 V=800.0 PL=0
MOVL C00685 V=800.0 PL=0
MOVL C00686 V=800.0 PL=0
MOVL C00687 V=800.0 PL=0
MOVL C00688 V=800.0 PL=0
MOVL C00689 V=800.0 PL=0
MOVL C00690 V=800.0 PL=0
MOVL C00691 V=800.0 PL=0
MOVL C00692 V=800.0 PL=0
MOVL C00693 V=800.0 PL=0
MOVL C00694 V=800.0 PL=0
MOVL C00695 V=800.0 PL=0
MOVL C00696 V=800.0 PL=0
MOVL C00697 V=800.0 PL=0
MOVL C00698 V=800.0 PL=0
MOVL C00699 V=800.0 PL=0
MOVL C00700 V=800.0 PL=0
MOVL C00701 V=800.0 PL=0
MOVL C00702 V=800.0 PL=0
MOVL C00703 V=800.0 PL=0
MOVL C00704 V=800.0 PL=0
MOVL C00705 V=800.0 PL=0
MOVL C00706 V=800.0 PL=0
MOVL C00707 V=800.0 PL=0
MOVL C00708 V=800.0 PL=0
MOVL C00709 V=800.0 PL=0
MOVL C00710 V=800.0 PL=0
MOVL C00711 V=800.0 PL=0
MOVL C00712 V=800.0 PL=0
MOVL C00713 V=800.0 PL=0
MOVL C00714 V=800.0 PL=0
MOVL C00715 V=800.0 PL=0
MOVL C00716 V=800.0 PL=0
MOVL C00717 V=800.0 PL=0
MOVL C00718 V=800.0 PL=0
MOVL C00719 V=800.0 PL=0
MOVL C00720 V=800.0 PL=0
MOVL C00721 V=800.0 PL=0
MOVL C00722 V=800.0 PL=0
MOVL C00723 V=800.0 PL=0
MOVL C00724 V=800.0 PL=0
MOVL C00725 V=800.0 PL=0
MOVL C00726 V=800.0 PL=0
MOVL C00727 V=800.0 PL=0
MOVL C00728 V=800.0 PL=0
MOVL C00729 V=800.0 PL=0
MOVL C00730 V=800.0 PL=0
MOVL C00731 V=800.0 PL=0
MOVL C00732 V=800.0 PL=0
MOVL C00733 V=800.0 PL=0
MOVL C00734 V=800.0 PL=0
MOVL C00735 V=800.0 PL=0
MOVL C00736 V=800.0 PL=0
MOVL C00737 V=800.0 PL=0
MOVL C00738 V=800.0 PL=0
MOVL C00739 V=800.0 PL=0
MOVL C00740 V=800.0 PL=0
MOVL C00741 V=800.0 PL=0
MOVL C00742 V=800.0 PL=0
MOVL C00743 V=800.0 PL=0
MOVL C00744 V=800.0 PL=0
MOVL C00745 V=800.0 PL=0
MOVL C00746 V=800.0 PL=0
MOVL C00747 V=800.0 PL=0
MOVL C00748 V=800.0 PL=0
MOVL C00749 V=800.0 PL=0
MOVL C00750 V=800.0 PL=0
MOVL C00751 V=800.0 PL=0
MOVL C00752 V=800.0 PL=0
MOVL C00753 V=800.0 PL=0
MOVL C00754 V=800.0 PL=0
MOVL C00755 V=800.0 PL=0
MOVL C00756 V=800.0 PL=0
MOVL C00757 V=800.0 PL=0
MOVL C00758 V=800.0 PL=0
MOVL C00759 V=800.0 PL=0
MOVL C00760 V=800.0 PL=0
MOVL C00761 V=800.0 PL=0
MOVL C00762 V=800.0 PL=0
MOVL C00763 V=800.0 PL=0
MOVL C00764 V=800.0 PL=0
MOVL C00765 V=800.0 PL=0
MOVL C00766 V=800.0 PL=0
MOVL C00767 V=800.0 PL=0
MOVL C00768 V=800.0 PL=0
MOVL C00769 V=800.0 PL=0
MOVL C00770 V=800.0 PL=0
MOVL C00771 V=800.0 PL=0
MOVL C00772 V=800.0 PL=0
MOVL C00773 V=800.0 PL=0
MOVL C00774 V=800.0 PL=0
MOVL C00775 V=800.0 PL=0
MOVL C00776 V=800.0 PL=0
MOVL C00777 V=800.0 PL=0
MOVL C00778 V=800.0 PL=0
MOVL C00779 V=800.0 PL=0
MOVL C00780 V=800.0 PL=0
MOVL C00781 V=800.0 PL=0
MOVL C00782 V=800.0 PL=0
MOVL C00783 V=800.0 PL=0
MOVL C00784 V=800.0 PL=0
MOVL C00785 V=800.0 PL=0
MOVL C00786 V=800.0 PL=0
MOVL C00787 V=800.0 PL=0
MOVL C00788 V=800.0 PL=0
MOVL C00789 V=800.0 PL=0
MOVL C00790 V=800.0 PL=0
MOVL C00791 V=800.0 PL=0
MOVL C00792 V=800.0 PL=0
MOVL C00793 V=800.0 PL=0
MOVL C00794 V=800.0 PL=0
MOVL C00795 V=800.0 PL=0
MOVL C00796 V=800.0 PL=0
MOVL C00797 V=800.0 PL=0
MOVL C00798 V=800.0 PL=0
MOVL C00799 V=800.0 PL=0
MOVL C00800 V=800.0 PL=0
MOVL C00801 V=800.0 PL=0
MOVL C00802 V=800.0 PL=0
MOVL C00803 V=800.0 PL=0
MOVL C00804 V=800.0 PL=0
MOVL C00805 V=800.0 PL=0
MOVL C00806 V=800.0 PL=0
MOVL C00807 V=800.0 PL=0
MOVL C00808 V=800.0 PL=0
MOVL C00809 V=800.0 PL=0
MOVL C00810 V=800.0 PL=0
MOVL C00811 V=800.0 PL=0
MOVL C00812 V=800.0 PL=0
MOVL C00813 V=800.0 PL=0
MOVL C00814 V=800.0 PL=0
MOVL C00815 V=800.0 PL=0
MOVL C00816 V=800.0 PL=0
MOVL C00817 V=800.0 PL=0
MOVL C00818 V=800.0 PL=0
MOVL C00819 V=800.0 PL=0
MOVL C00820 V=800.0 PL=0
MOVL C00821 V=800.0 PL=0
MOVL C00822 V=800.0 PL=0
MOVL C00823 V=800.0 PL=0
MOVL C00824 V=800.0 PL=0
MOVL C00825 V=800.0 PL=0
MOVL C00826 V=800.0 PL=0
MOVL C00827 V=800.0 PL=0
MOVL C00828 V=800.0 PL=0
MOVL C00829 V=800.0 PL=0
MOVL C00830 V=800.0 PL=0
MOVL C00831 V=800.0 PL=0
MOVL C00832 V=800.0 PL=0
MOVL C00833 V=800.0 PL=0
MOVL C00834 V=800.0 PL=0
MOVL C00835 V=800.0 PL=0
MOVL C00836 V=800.0 PL=0
MOVL C00837 V=800.0 PL=0
MOVL C00838 V=800.0 PL=0
MOVL C00839 V=800.0 PL=0
MOVL C00840 V=800.0 PL=0
MOVL C00841 V=800.0 PL=0
MOVL C00842 V=800.0 PL=0
MOVL C00843 V=800.0 PL=0
MOVL C00844 V=800.0 PL=0
MOVL C00845 V=800.0 PL=0
MOVL C00846 V=800.0 PL=0
MOVL C00847 V=800.0 PL=0
MOVL C00848 V=800.0 PL=0
MOVL C00849 V=800.0 PL=0
MOVL C00850 V=800.0 PL=0
MOVL C00851 V=800.0 PL=0
MOVL C00852 V=800.0 PL=0
MOVL C00853 V=800.0 PL=0
MOVL C00854 V=800.0 PL=0
MOVL C00855 V=800.0 PL=0
MOVL C00856 V=800.0 PL=0
MOVL C00857 V=800.0 PL=0
MOVL C00858 V=800.0 PL=0
MOVL C00859 V=800.0 PL=0
MOVL C00860 V=800.0 PL=0
MOVL C00861 V=800.0 PL=0
MOVL C00862 V=800.0 PL=0
MOVL C00863 V=800.0 PL=0
MOVL C00864 V=800.0 PL=0
MOVL C00865 V=800.0 PL=0
MOVL C00866 V=800.0 PL=0
MOVL C00867 V=800.0 PL=0
MOVL C00868 V=800.0 PL=0
MOVL C00869 V=800.0 PL=0
MOVL C00870 V=800.0 PL=0
MOVL C00871 V=800.0 PL=0
MOVL C00872 V=800.0 PL=0
MOVL C00873 V=800.0 PL=0
MOVL C00874 V=800.0 PL=0
MOVL C00875 V=800.0 PL=0
MOVL C00876 V=800.0 PL=0
MOVL C00877 V=800.0 PL=0
MOVL C00878 V=800.0 PL=0
MOVL C00879 V=800.0 PL=0
MOVL C00880 V=800.0 PL=0
MOVL C00881 V=800.0 PL=0
MOVL C00882 V=800.0 PL=0
MOVL C00883 V=800.0 PL=0
MOVL C00884 V=800.0 PL=0
MOVL C00885 V=800.0 PL=0
MOVL C00886 V=800.0 PL=0
MOVL C00887 V=800.0 PL=0
MOVL C00888 V=800.0 PL=0
MOVL C00889 V=800.0 PL=0
MOVL C00890 V=800.0 PL=0
MOVL C00891 V=800.0 PL=0
MOVL C00892 V=800.0 PL=0
MOVL C00893 V=800.0 PL=0
MOVL C00894 V=800.0 PL=0
MOVL C00895 V=800.0 PL=0
MOVL C00896 V=800.0 PL=0
MOVL C00897 V=800.0 PL=0
MOVL C00898 V=800.0 PL=0
MOVL C00899 V=800.0 PL=0
MOVL C00900 V=800.0 PL=0
MOVL C00901 V=800.0 PL=0
MOVL C00902 V=800.0 PL=0
MOVL C00903 V=800.0 PL=0
MOVL C00904 V=800.0 PL=0
MOVL C00905 V=800.0 PL=0
MOVL C00906 V=800.0 PL=0
MOVL C00907 V=800.0 PL=0
MOVL C00908 V=800.0 PL=0
MOVL C00909 V=800.0 PL=0
MOVL C00910 V=800.0 PL=0
MOVL C00911 V=800.0 PL=0
MOVL C00912 V=800.0 PL=0
MOVL C00913 V=800.0 PL=0
MOVL C00914 V=800.0 PL=0
MOVL C00915 V=800.0 PL=0
MOVL C00916 V=800.0 PL=0
MOVL C00917 V=800.0 PL=0
MOVL C00918 V=800.0 PL=0
MOVL C00919 V=800.0 PL=0
MOVL C00920 V=800.0 PL=0
MOVL C00921 V=800.0 PL=0
MOVL C00922 V=800.0 PL=0
MOVL C00923 V=800.0 PL=0
MOVL C00924 V=800.0 PL=0
MOVL C00925 V=800.0 PL=0
MOVL C00926 V=800.0 PL=0
MOVL C00927 V=800.0 PL=0
MOVL C00928 V=800.0 PL=0
MOVL C00929 V=800.0 PL=0
MOVL C00930 V=800.0 PL=0
MOVL C00931 V=800.0 PL=0
MOVL C00932 V=800.0 PL=0
MOVL C00933 V=800.0 PL=0
MOVL C00934 V=800.0 PL=0
MOVL C00935 V=800.0 PL=0
MOVL C00936 V=800.0 PL=0
MOVL C00937 V=800.0 PL=0
MOVL C00938 V=800.0 PL=0
MOVL C00939 V=800.0 PL=0
MOVL C00940 V=800.0 PL=0
MOVL C00941 V=800.0 PL=0
MOVL C00942 V=800.0 PL=0
MOVL C00943 V=800.0 PL=0
MOVL C00944 V=800.0 PL=0
MOVL C00945 V=800.0 PL=0
MOVL C00946 V=800.0 PL=0
MOVL C00947 V=800.0 PL=0
MOVL C00948 V=800.0 PL=0
MOVL C00949 V=800.0 PL=0
MOVL C00950 V=800.0 PL=0
MOVL C00951 V=800.0 PL=0
MOVL C00952 V=800.0 PL=0
MOVL C00953 V=800.0 PL=0
MOVL C00954 V=800.0 PL=0
MOVL C00955 V=800.0 PL=0
MOVL C00956 V=800.0 PL=0
MOVL C00957 V=800.0 PL=0
MOVL C00958 V=800.0 PL=0
MOVL C00959 V=800.0 PL=0
MOVL C00960 V=800.0 PL=0
MOVL C00961 V=800.0 PL=0
MOVL C00962 V=800.0 PL=0
MOVL C00963 V=800.0 PL=0
MOVL C00964 V=800.0 PL=0
MOVL C00965 V=800.0 PL=0
MOVL C00966 V=800.0 PL=0
MOVL C00967 V=800.0 PL=0
MOVL C00968 V=800.0 PL=0
MOVL C00969 V=800.0 PL=0
MOVL C00970 V=800.0 PL=0
MOVL C00971 V=800.0 PL=0
MOVL C00972 V=800.0 PL=0
MOVL C00973 V=800.0 PL=0
MOVL C00974 V=800.0 PL=0
MOVL C00975 V=800.0 PL=0
MOVL C00976 V=800.0 PL=0
MOVL C00977 V=800.0 PL=0
MOVL C00978 V=800.0 PL=0
MOVL C00979 V=800.0 PL=0
MOVL C00980 V=800.0 PL=0
MOVL C00981 V=800.0 PL=0
MOVL C00982 V=800.0 PL=0
MOVL C00983 V=800.0 PL=0
MOVL C00984 V=800.0 PL=0
MOVL C00985 V=800.0 PL=0
MOVL C00986 V=800.0 PL=0
MOVL C00987 V=800.0 PL=0
MOVL C00988 V=800.0 PL=0
MOVL C00989 V=800.0 PL=0
MOVL C00990 V=800.0 PL=0
MOVL C00991 V=800.0 PL=0
MOVL C00992 V=800.0 PL=0
MOVL C00993 V=800.0 PL=0
MOVL C00994 V=800.0 PL=0
MOVL C00995 V=800.0 PL=0
MOVL C00996 V=800.0 PL=0
MOVL C00997 V=800.0 PL=0
MOVL C00998 V=800.0 PL=0
MOVL C00999 V=800.0 PL=0
MOVL C01000 V=800.0 PL=0
MOVL C01001 V=800.0 PL=0
MOVL C01002 V=800.0 PL=0
MOVL C01003 V=800.0 PL=0
MOVL C01004 V=800.0 PL=0
MOVL C01005 V=800.0 PL=0
MOVL C01006 V=800.0 PL=0
MOVL C01007 V=800.0 PL=0
MOVL C01008 V=800.0 PL=0
MOVL C01009 V=800.0 PL=0
MOVL C01010 V=800.0 PL=0
MOVL C01011 V=800.0 PL=0
MOVL C01012 V=800.0 PL=0
MOVL C01013 V=800.0 PL=0
MOVL C01014 V=800.0 PL=0
MOVL C01015 V=800.0 PL=0
MOVL C01016 V=800.0 PL=0
MOVL C01017 V=800.0 PL=0
MOVL C01018 V=800.0 PL=0
MOVL C01019 V=800.0 PL=0
MOVL C01020 V=800.0 PL=0
MOVL C01021 V=800.0 PL=0
MOVL C01022 V=800.0 PL=0
MOVL C01023 V=800.0 PL=0
MOVL C01024 V=800.0 PL=0
MOVL C01025 V=800.0 PL=0
MOVL C01026 V=800.0 PL=0
MOVL C01027 V=800.0 PL=0
MOVL C01028 V=800.0 PL=0
MOVL C01029 V=800.0 PL=0
MOVL C01030 V=800.0 PL=0
MOVL C01031 V=800.0 PL=0
MOVL C01032 V=800.0 PL=0
MOVL C01033 V=800.0 PL=0
MOVL C01034 V=800.0 PL=0
MOVL C01035 V=800.0 PL=0
MOVL C01036 V=800.0 PL=0
MOVL C01037 V=800.0 PL=0
MOVL C01038 V=800.0 PL=0
MOVL C01039 V=800.0 PL=0
MOVL C01040 V=800.0 PL=0
MOVL C01041 V=800.0 PL=0
MOVL C01042 V=800.0 PL=0
MOVL C01043 V=800.0 PL=0
MOVL C01044 V=800.0 PL=0
MOVL C01045 V=800.0 PL=0
MOVL C01046 V=800.0 PL=0
MOVL C01047 V=800.0 PL=0
MOVL C01048 V=800.0 PL=0
MOVL C01049 V=800.0 PL=0
MOVL C01050 V=800.0 PL=0
MOVL C01051 V=800.0 PL=0
MOVL C01052 V=800.0 PL=0
MOVL C01053 V=800.0 PL=0
MOVL C01054 V=800.0 PL=0
MOVL C01055 V=800.0 PL=0
MOVL C01056 V=800.0 PL=0
MOVL C01057 V=800.0 PL=0
MOVL C01058 V=800.0 PL=0
MOVL C01059 V=800.0 PL=0
MOVL C01060 V=800.0 PL=0
MOVL C01061 V=800.0 PL=0
MOVL C01062 V=800.0 PL=0
MOVL C01063 V=800.0 PL=0
MOVL C01064 V=800.0 PL=0
MOVL C01065 V=800.0 PL=0
MOVL C01066 V=800.0 PL=0
MOVL C01067 V=800.0 PL=0
MOVL C01068 V=800.0 PL=0
MOVL C01069 V=800.0 PL=0
MOVL C01070 V=800.0 PL=0
MOVL C01071 V=800.0 PL=0
MOVL C01072 V=800.0 PL=0
MOVL C01073 V=800.0 PL=0
MOVL C01074 V=800.0 PL=0
MOVL C01075 V=800.0 PL=0
MOVL C01076 V=800.0 PL=0
MOVL C01077 V=800.0 PL=0
MOVL C01078 V=800.0 PL=0
MOVL C01079 V=800.0 PL=0
MOVL C01080 V=800.0 PL=0
MOVL C01081 V=800.0 PL=0
MOVL C01082 V=800.0 PL=0
MOVL C01083 V=800.0 PL=0
MOVL C01084 V=800.0 PL=0
MOVL C01085 V=800.0 PL=0
MOVL C01086 V=800.0 PL=0
MOVL C01087 V=800.0 PL=0
MOVL C01088 V=800.0 PL=0
MOVL C01089 V=800.0 PL=0
MOVL C01090 V=800.0 PL=0
MOVL C01091 V=800.0 PL=0
MOVL C01092 V=800.0 PL=0
MOVL C01093 V=800.0 PL=0
MOVL C01094 V=800.0 PL=0
MOVL C01095 V=800.0 PL=0
MOVL C01096 V=800.0 PL=0
MOVL C01097 V=800.0 PL=0
MOVL C01098 V=800.0 PL=0
MOVL C01099 V=800.0 PL=0
MOVL C01100 V=800.0 PL=0
MOVL C01101 V=800.0 PL=0
MOVL C01102 V=800.0 PL=0
MOVL C01103 V=800.0 PL=0
MOVL C01104 V=800.0 PL=0
MOVL C01105 V=800.0 PL=0
MOVL C01106 V=800.0 PL=0
MOVL C01107 V=800.0 PL=0
MOVL C01108 V=800.0 PL=0
MOVL C01109 V=800.0 PL=0
MOVL C01110 V=800.0 PL=0
MOVL C01111 V=800.0 PL=0
MOVL C01112 V=800.0 PL=0
MOVL C01113 V=800.0 PL=0
MOVL C01114 V=800.0 PL=0
MOVL C01115 V=800.0 PL=0
MOVL C01116 V=800.0 PL=0
MOVL C01117 V=800.0 PL=0
MOVL C01118 V=800.0 PL=0
MOVL C01119 V=800.0 PL=0
MOVL C01120 V=800.0 PL=0
MOVL C01121 V=800.0 PL=0
MOVL C01122 V=800.0 PL=0
MOVL C01123 V=800.0 PL=0
MOVL C01124 V=800.0 PL=0
MOVL C01125 V=800.0 PL=0
MOVL C01126 V=800.0 PL=0
MOVL C01127 V=800.0 PL=0
MOVL C01128 V=800.0 PL=0
MOVL C01129 V=800.0 PL=0
MOVL C01130 V=800.0 PL=0
MOVL C01131 V=800.0 PL=0
MOVL C01132 V=800.0 PL=0
MOVL C01133 V=800.0 PL=0
MOVL C01134 V=800.0 PL=0
MOVL C01135 V=800.0 PL=0
MOVL C01136 V=800.0 PL=0
MOVL C01137 V=800.0 PL=0
MOVL C01138 V=800.0 PL=0
MOVL C01139 V=800.0 PL=0
MOVL C01140 V=800.0 PL=0
MOVL C01141 V=800.0 PL=0
MOVL C01142 V=800.0 PL=0
MOVL C01143 V=800.0 PL=0
MOVL C01144 V=800.0 PL=0
MOVL C01145 V=800.0 PL=0
MOVL C01146 V=800.0 PL=0
MOVL C01147 V=800.0 PL=0
MOVL C01148 V=800.0 PL=0
MOVL C01149 V=800.0 PL=0
MOVL C01150 V=800.0 PL=0
MOVL C01151 V=800.0 PL=0
MOVL C01152 V=800.0 PL=0
MOVL C01153 V=800.0 PL=0
MOVL C01154 V=800.0 PL=0
MOVL C01155 V=800.0 PL=0
MOVL C01156 V=800.0 PL=0
MOVL C01157 V=800.0 PL=0
MOVL C01158 V=800.0 PL=0
MOVL C01159 V=800.0 PL=0
MOVL C01160 V=800.0 PL=0
MOVL C01161 V=800.0 PL=0
MOVL C01162 V=800.0 PL=0
MOVL C01163 V=800.0 PL=0
MOVL C01164 V=800.0 PL=0
MOVL C01165 V=800.0 PL=0
MOVL C01166 V=800.0 PL=0
MOVL C01167 V=800.0 PL=0
MOVL C01168 V=800.0 PL=0
MOVL C01169 V=800.0 PL=0
MOVL C01170 V=800.0 PL=0
MOVL C01171 V=800.0 PL=0
MOVL C01172 V=800.0 PL=0
MOVL C01173 V=800.0 PL=0
MOVL C01174 V=800.0 PL=0
MOVL C01175 V=800.0 PL=0
MOVL C01176 V=800.0 PL=0
MOVL C01177 V=800.0 PL=0
MOVL C01178 V=800.0 PL=0
MOVL C01179 V=800.0 PL=0
MOVL C01180 V=800.0 PL=0
MOVL C01181 V=800.0 PL=0
MOVL C01182 V=800.0 PL=0
MOVL C01183 V=800.0 PL=0
MOVL C01184 V=800.0 PL=0
MOVL C01185 V=800.0 PL=0
MOVL C01186 V=800.0 PL=0
MOVL C01187 V=800.0 PL=0
MOVL C01188 V=800.0 PL=0
MOVL C01189 V=800.0 PL=0
MOVL C01190 V=800.0 PL=0
MOVL C01191 V=800.0 PL=0
MOVL C01192 V=800.0 PL=0
MOVL C01193 V=800.0 PL=0
MOVL C01194 V=800.0 PL=0
MOVL C01195 V=800.0 PL=0
MOVL C01196 V=800.0 PL=0
MOVL C01197 V=800.0 PL=0
MOVL C01198 V=800.0 PL=0
MOVL C01199 V=800.0 PL=0
MOVL C01200 V=800.0 PL=0
MOVL C01201 V=800.0 PL=0
MOVL C01202 V=800.0 PL=0
MOVL C01203 V=800.0 PL=0
MOVL C01204 V=800.0 PL=0
MOVL C01205 V=800.0 PL=0
MOVL C01206 V=800.0 PL=0
MOVL C01207 V=800.0 PL=0
MOVL C01208 V=800.0 PL=0
MOVL C01209 V=800.0 PL=0
MOVL C01210 V=800.0 PL=0
MOVL C01211 V=800.0 PL=0
MOVL C01212 V=800.0 PL=0
MOVL C01213 V=800.0 PL=0
MOVL C01214 V=800.0 PL=0
MOVL C01215 V=800.0 PL=0
MOVL C01216 V=800.0 PL=0
MOVL C01217 V=800.0 PL=0
MOVL C01218 V=800.0 PL=0
MOVL C01219 V=800.0 PL=0
MOVL C01220 V=800.0 PL=0
MOVL C01221 V=800.0 PL=0
MOVL C01222 V=800.0 PL=0
MOVL C01223 V=800.0 PL=0
MOVL C01224 V=800.0 PL=0
MOVL C01225 V=800.0 PL=0
MOVL C01226 V=800.0 PL=0
MOVL C01227 V=800.0 PL=0
MOVL C01228 V=800.0 PL=0
MOVL C01229 V=800.0 PL=0
MOVL C01230 V=800.0 PL=0
MOVL C01231 V=800.0 PL=0
MOVL C01232 V=800.0 PL=0
MOVL C01233 V=800.0 PL=0
MOVL C01234 V=800.0 PL=0
MOVL C01235 V=800.0 PL=0
MOVL C01236 V=800.0 PL=0
MOVL C01237 V=800.0 PL=0
MOVL C01238 V=800.0 PL=0
MOVL C01239 V=800.0 PL=0
MOVL C01240 V=800.0 PL=0
MOVL C01241 V=800.0 PL=0
MOVL C01242 V=800.0 PL=0
MOVL C01243 V=800.0 PL=0
MOVL C01244 V=800.0 PL=0
MOVL C01245 V=800.0 PL=0
MOVL C01246 V=800.0 PL=0
MOVL C01247 V=800.0 PL=0
MOVL C01248 V=800.0 PL=0
MOVL C01249 V=800.0 PL=0
MOVL C01250 V=800.0 PL=0
MOVL C01251 V=800.0 PL=0
MOVL C01252 V=800.0 PL=0
MOVL C01253 V=800.0 PL=0
MOVL C01254 V=800.0 PL=0
MOVL C01255 V=800.0 PL=0
MOVL C01256 V=800.0 PL=0
MOVL C01257 V=800.0 PL=0
MOVL C01258 V=800.0 PL=0
MOVL C01259 V=800.0 PL=0
MOVL C01260 V=800.0 PL=0
MOVL C01261 V=800.0 PL=0
MOVL C01262 V=800.0 PL=0
MOVL C01263 V=800.0 PL=0
MOVL C01264 V=800.0 PL=0
MOVL C01265 V=800.0 PL=0
MOVL C01266 V=800.0 PL=0
MOVL C01267 V=800.0 PL=0
MOVL C01268 V=800.0 PL=0
MOVL C01269 V=800.0 PL=0
MOVL C01270 V=800.0 PL=0
MOVL C01271 V=800.0 PL=0
MOVL C01272 V=800.0 PL=0
MOVL C01273 V=800.0 PL=0
MOVL C01274 V=800.0 PL=0
MOVL C01275 V=800.0 PL=0
MOVL C01276 V=800.0 PL=0
MOVL C01277 V=800.0 PL=0
MOVL C01278 V=800.0 PL=0
MOVL C01279 V=800.0 PL=0
MOVL C01280 V=800.0 PL=0
MOVL C01281 V=800.0 PL=0
MOVL C01282 V=800.0 PL=0
MOVL C01283 V=800.0 PL=0
MOVL C01284 V=800.0 PL=0
MOVL C01285 V=800.0 PL=0
MOVL C01286 V=800.0 PL=0
MOVL C01287 V=800.0 PL=0
MOVL C01288 V=800.0 PL=0
MOVL C01289 V=800.0 PL=0
MOVL C01290 V=800.0 PL=0
MOVL C01291 V=800.0 PL=0
MOVL C01292 V=800.0 PL=0
MOVL C01293 V=800.0 PL=0
MOVL C01294 V=800.0 PL=0
MOVL C01295 V=800.0 PL=0
MOVL C01296 V=800.0 PL=0
MOVL C01297 V=800.0 PL=0
MOVL C01298 V=800.0 PL=0
MOVL C01299 V=800.0 PL=0
MOVL C01300 V=800.0 PL=0
MOVL C01301 V=800.0 PL=0
MOVL C01302 V=800.0 PL=0
MOVL C01303 V=800.0 PL=0
MOVL C01304 V=800.0 PL=0
MOVL C01305 V=800.0 PL=0
MOVL C01306 V=800.0 PL=0
MOVL C01307 V=800.0 PL=0
MOVL C01308 V=800.0 PL=0
MOVL C01309 V=800.0 PL=0
MOVL C01310 V=800.0 PL=0
MOVL C01311 V=800.0 PL=0
MOVL C01312 V=800.0 PL=0
MOVL C01313 V=800.0 PL=0
MOVL C01314 V=800.0 PL=0
MOVL C01315 V=800.0 PL=0
MOVL C01316 V=800.0 PL=0
MOVL C01317 V=800.0 PL=0
MOVL C01318 V=800.0 PL=0
MOVL C01319 V=800.0 PL=0
MOVL C01320 V=800.0 PL=0
MOVL C01321 V=800.0 PL=0
MOVL C01322 V=800.0 PL=0
MOVL C01323 V=800.0 PL=0
MOVL C01324 V=800.0 PL=0
MOVL C01325 V=800.0 PL=0
MOVL C01326 V=800.0 PL=0
MOVL C01327 V=800.0 PL=0
MOVL C01328 V=800.0 PL=0
MOVL C01329 V=800.0 PL=0
MOVL C01330 V=800.0 PL=0
MOVL C01331 V=800.0 PL=0
MOVL C01332 V=800.0 PL=0
MOVL C01333 V=800.0 PL=0
MOVL C01334 V=800.0 PL=0
MOVL C01335 V=800.0 PL=0
MOVL C01336 V=800.0 PL=0
MOVL C01337 V=800.0 PL=0
MOVL C01338 V=800.0 PL=0
MOVL C01339 V=800.0 PL=0
MOVL C01340 V=800.0 PL=0
MOVL C01341 V=800.0 PL=0
MOVL C01342 V=800.0 PL=0
MOVL C01343 V=800.0 PL=0
MOVL C01344 V=800.0 PL=0
MOVL C01345 V=800.0 PL=0
MOVL C01346 V=800.0 PL=0
MOVL C01347 V=800.0 PL=0
MOVL C01348 V=800.0 PL=0
MOVL C01349 V=800.0 PL=0
MOVL C01350 V=800.0 PL=0
MOVL C01351 V=800.0 PL=0
MOVL C01352 V=800.0 PL=0
MOVL C01353 V=800.0 PL=0
MOVL C01354 V=800.0 PL=0
MOVL C01355 V=800.0 PL=0
MOVL C01356 V=800.0 PL=0
MOVL C01357 V=800.0 PL=0
MOVL C01358 V=800.0 PL=0
MOVL C01359 V=800.0 PL=0
MOVL C01360 V=800.0 PL=0
MOVL C01361 V=800.0 PL=0
MOVL C01362 V=800.0 PL=0
MOVL C01363 V=800.0 PL=0
MOVL C01364 V=800.0 PL=0
MOVL C01365 V=800.0 PL=0
MOVL C01366 V=800.0 PL=0
MOVL C01367 V=800.0 PL=0
MOVL C01368 V=800.0 PL=0
MOVL C01369 V=800.0 PL=0
MOVL C01370 V=800.0 PL=0
MOVL C01371 V=800.0 PL=0
MOVL C01372 V=800.0 PL=0
MOVL C01373 V=800.0 PL=0
MOVL C01374 V=800.0 PL=0
MOVL C01375 V=800.0 PL=0
MOVL C01376 V=800.0 PL=0
MOVL C01377 V=800.0 PL=0
MOVL C01378 V=800.0 PL=0
MOVL C01379 V=800.0 PL=0
MOVL C01380 V=800.0 PL=0
MOVL C01381 V=800.0 PL=0
MOVL C01382 V=800.0 PL=0
MOVL C01383 V=800.0 PL=0
MOVL C01384 V=800.0 PL=0
MOVL C01385 V=800.0 PL=0
MOVL C01386 V=800.0 PL=0
MOVL C01387 V=800.0 PL=0
MOVL C01388 V=800.0 PL=0
MOVL C01389 V=800.0 PL=0
MOVL C01390 V=800.0 PL=0
MOVL C01391 V=800.0 PL=0
MOVL C01392 V=800.0 PL=0
MOVL C01393 V=800.0 PL=0
MOVL C01394 V=800.0 PL=0
MOVL C01395 V=800.0 PL=0
MOVL C01396 V=800.0 PL=0
MOVL C01397 V=800.0 PL=0
MOVL C01398 V=800.0 PL=0
MOVL C01399 V=800.0 PL=0
MOVL C01400 V=800.0 PL=0
MOVL C01401 V=800.0 PL=0
MOVL C01402 V=800.0 PL=0
MOVL C01403 V=800.0 PL=0
MOVL C01404 V=800.0 PL=0
MOVL C01405 V=800.0 PL=0
MOVL C01406 V=800.0 PL=0
MOVL C01407 V=800.0 PL=0
MOVL C01408 V=800.0 PL=0
MOVL C01409 V=800.0 PL=0
MOVL C01410 V=800.0 PL=0
MOVL C01411 V=800.0 PL=0
MOVL C01412 V=800.0 PL=0
MOVL C01413 V=800.0 PL=0
MOVL C01414 V=800.0 PL=0
MOVL C01415 V=800.0 PL=0
MOVL C01416 V=800.0 PL=0
MOVL C01417 V=800.0 PL=0
MOVL C01418 V=800.0 PL=0
MOVL C01419 V=800.0 PL=0
MOVL C01420 V=800.0 PL=0
MOVL C01421 V=800.0 PL=0
MOVL C01422 V=800.0 PL=0
MOVL C01423 V=800.0 PL=0
MOVL C01424 V=800.0 PL=0
MOVL C01425 V=800.0 PL=0
MOVL C01426 V=800.0 PL=0
MOVL C01427 V=800.0 PL=0
MOVL C01428 V=800.0 PL=0
MOVL C01429 V=800.0 PL=0
MOVL C01430 V=800.0 PL=0
MOVL C01431 V=800.0 PL=0
MOVL C01432 V=800.0 PL=0
MOVL C01433 V=800.0 PL=0
MOVL C01434 V=800.0 PL=0
MOVL C01435 V=800.0 PL=0
MOVL C01436 V=800.0 PL=0
MOVL C01437 V=800.0 PL=0
MOVL C01438 V=800.0 PL=0
MOVL C01439 V=800.0 PL=0
MOVL C01440 V=800.0 PL=0
MOVL C01441 V=800.0 PL=0
MOVL C01442 V=800.0 PL=0
MOVL C01443 V=800.0 PL=0
MOVL C01444 V=800.0 PL=0
MOVL C01445 V=800.0 PL=0
MOVL C01446 V=800.0 PL=0
MOVL C01447 V=800.0 PL=0
MOVL C01448 V=800.0 PL=0
MOVL C01449 V=800.0 PL=0
MOVL C01450 V=800.0 PL=0
MOVL C01451 V=800.0 PL=0
MOVL C01452 V=800.0 PL=0
MOVL C01453 V=800.0 PL=0
MOVL C01454 V=800.0 PL=0
MOVL C01455 V=800.0 PL=0
MOVL C01456 V=800.0 PL=0
MOVL C01457 V=800.0 PL=0
MOVL C01458 V=800.0 PL=0
MOVL C01459 V=800.0 PL=0
MOVL C01460 V=800.0 PL=0
MOVL C01461 V=800.0 PL=0
MOVL C01462 V=800.0 PL=0
MOVL C01463 V=800.0 PL=0
MOVL C01464 V=800.0 PL=0
MOVL C01465 V=800.0 PL=0
MOVL C01466 V=800.0 PL=0
MOVL C01467 V=800.0 PL=0
MOVL C01468 V=800.0 PL=0
MOVL C01469 V=800.0 PL=0
MOVL C01470 V=800.0 PL=0
MOVL C01471 V=800.0 PL=0
MOVL C01472 V=800.0 PL=0
MOVL C01473 V=800.0 PL=0
MOVL C01474 V=800.0 PL=0
MOVL C01475 V=800.0 PL=0
MOVL C01476 V=800.0 PL=0
MOVL C01477 V=800.0 PL=0
MOVL C01478 V=800.0 PL=0
MOVL C01479 V=800.0 PL=0
MOVL C01480 V=800.0 PL=0
MOVL C01481 V=800.0 PL=0
MOVL C01482 V=800.0 PL=0
MOVL C01483 V=800.0 PL=0
MOVL C01484 V=800.0 PL=0
MOVL C01485 V=800.0 PL=0
MOVL C01486 V=800.0 PL=0
MOVL C01487 V=800.0 PL=0
MOVL C01488 V=800.0 PL=0
MOVL C01489 V=800.0 PL=0
MOVL C01490 V=800.0 PL=0
MOVL C01491 V=800.0 PL=0
MOVL C01492 V=800.0 PL=0
MOVL C01493 V=800.0 PL=0
MOVL C01494 V=800.0 PL=0
MOVL C01495 V=800.0 PL=0
MOVL C01496 V=800.0 PL=0
MOVL C01497 V=800.0 PL=0
MOVL C01498 V=800.0 PL=0
MOVL C01499 V=800.0 PL=0
MOVL C01500 V=800.0 PL=0
MOVL C01501 V=800.0 PL=0
MOVL C01502 V=800.0 PL=0
MOVL C01503 V=800.0 PL=0
MOVL C01504 V=800.0 PL=0
MOVL C01505 V=800.0 PL=0
MOVL C01506 V=800.0 PL=0
MOVL C01507 V=800.0 PL=0
MOVL C01508 V=800.0 PL=0
MOVL C01509 V=800.0 PL=0
MOVL C01510 V=800.0 PL=0
MOVL C01511 V=800.0 PL=0
MOVL C01512 V=800.0 PL=0
MOVL C01513 V=800.0 PL=0
MOVL C01514 V=800.0 PL=0
MOVL C01515 V=800.0 PL=0
MOVL C01516 V=800.0 PL=0
MOVL C01517 V=800.0 PL=0
MOVL C01518 V=800.0 PL=0
MOVL C01519 V=800.0 PL=0
MOVL C01520 V=800.0 PL=0
MOVL C01521 V=800.0 PL=0
MOVL C01522 V=800.0 PL=0
MOVL C01523 V=800.0 PL=0
MOVL C01524 V=800.0 PL=0
MOVL C01525 V=800.0 PL=0
MOVL C01526 V=800.0 PL=0
MOVL C01527 V=800.0 PL=0
MOVL C01528 V=800.0 PL=0
MOVL C01529 V=800.0 PL=0
MOVL C01530 V=800.0 PL=0
MOVL C01531 V=800.0 PL=0
MOVL C01532 V=800.0 PL=0
MOVL C01533 V=800.0 PL=0
MOVL C01534 V=800.0 PL=0
MOVL C01535 V=800.0 PL=0
MOVL C01536 V=800.0 PL=0
MOVL C01537 V=800.0 PL=0
MOVL C01538 V=800.0 PL=0
MOVL C01539 V=800.0 PL=0
MOVL C01540 V=800.0 PL=0
MOVL C01541 V=800.0 PL=0
MOVL C01542 V=800.0 PL=0
MOVL C01543 V=800.0 PL=0
MOVL C01544 V=800.0 PL=0
MOVL C01545 V=800.0 PL=0
MOVL C01546 V=800.0 PL=0
MOVL C01547 V=800.0 PL=0
MOVL C01548 V=800.0 PL=0
MOVL C01549 V=800.0 PL=0
MOVL C01550 V=800.0 PL=0
MOVL C01551 V=800.0 PL=0
MOVL C01552 V=800.0 PL=0
MOVL C01553 V=800.0 PL=0
MOVL C01554 V=800.0 PL=0
MOVL C01555 V=800.0 PL=0
MOVL C01556 V=800.0 PL=0
MOVL C01557 V=800.0 PL=0
MOVL C01558 V=800.0 PL=0
MOVL C01559 V=800.0 PL=0
MOVL C01560 V=800.0 PL=0
MOVL C01561 V=800.0 PL=0
MOVL C01562 V=800.0 PL=0
MOVL C01563 V=800.0 PL=0
MOVL C01564 V=800.0 PL=0
MOVL C01565 V=800.0 PL=0
MOVL C01566 V=800.0 PL=0
MOVL C01567 V=800.0 PL=0
MOVL C01568 V=800.0 PL=0
MOVL C01569 V=800.0 PL=0
MOVL C01570 V=800.0 PL=0
MOVL C01571 V=800.0 PL=0
MOVL C01572 V=800.0 PL=0
MOVL C01573 V=800.0 PL=0
MOVL C01574 V=800.0 PL=0
MOVL C01575 V=800.0 PL=0
MOVL C01576 V=800.0 PL=0
MOVL C01577 V=800.0 PL=0
MOVL C01578 V=800.0 PL=0
MOVL C01579 V=800.0 PL=0
MOVL C01580 V=800.0 PL=0
MOVL C01581 V=800.0 PL=0
MOVL C01582 V=800.0 PL=0
MOVL C01583 V=800.0 PL=0
MOVL C01584 V=800.0 PL=0
MOVL C01585 V=800.0 PL=0
MOVL C01586 V=800.0 PL=0
MOVL C01587 V=800.0 PL=0
MOVL C01588 V=800.0 PL=0
MOVL C01589 V=800.0 PL=0
MOVL C01590 V=800.0 PL=0
MOVL C01591 V=800.0 PL=0
MOVL C01592 V=800.0 PL=0
MOVL C01593 V=800.0 PL=0
MOVL C01594 V=800.0 PL=0
MOVL C01595 V=800.0 PL=0
MOVL C01596 V=800.0 PL=0
MOVL C01597 V=800.0 PL=0
MOVL C01598 V=800.0 PL=0
MOVL C01599 V=800.0 PL=0
MOVL C01600 V=800.0 PL=0
MOVL C01601 V=800.0 PL=0
MOVL C01602 V=800.0 PL=0
MOVL C01603 V=800.0 PL=0
MOVL C01604 V=800.0 PL=0
MOVL C01605 V=800.0 PL=0
MOVL C01606 V=800.0 PL=0
MOVL C01607 V=800.0 PL=0
MOVL C01608 V=800.0 PL=0
MOVL C01609 V=800.0 PL=0
MOVL C01610 V=800.0 PL=0
MOVL C01611 V=800.0 PL=0
MOVL C01612 V=800.0 PL=0
MOVL C01613 V=800.0 PL=0
MOVL C01614 V=800.0 PL=0
MOVL C01615 V=800.0 PL=0
MOVL C01616 V=800.0 PL=0
MOVL C01617 V=800.0 PL=0
MOVL C01618 V=800.0 PL=0
MOVL C01619 V=800.0 PL=0
MOVL C01620 V=800.0 PL=0
MOVL C01621 V=800.0 PL=0
MOVL C01622 V=800.0 PL=0
MOVL C01623 V=800.0 PL=0
MOVL C01624 V=800.0 PL=0
MOVL C01625 V=800.0 PL=0
MOVL C01626 V=800.0 PL=0
MOVL C01627 V=800.0 PL=0
MOVL C01628 V=800.0 PL=0
MOVL C01629 V=800.0 PL=0
MOVL C01630 V=800.0 PL=0
MOVL C01631 V=800.0 PL=0
MOVL C01632 V=800.0 PL=0
MOVL C01633 V=800.0 PL=0
MOVL C01634 V=800.0 PL=0
MOVL C01635 V=800.0 PL=0
MOVL C01636 V=800.0 PL=0
MOVL C01637 V=800.0 PL=0
MOVL C01638 V=800.0 PL=0
MOVL C01639 V=800.0 PL=0
MOVL C01640 V=800.0 PL=0
MOVL C01641 V=800.0 PL=0
MOVL C01642 V=800.0 PL=0
MOVL C01643 V=800.0 PL=0
MOVL C01644 V=800.0 PL=0
MOVL C01645 V=800.0 PL=0
MOVL C01646 V=800.0 PL=0
MOVL C01647 V=800.0 PL=0
MOVL C01648 V=800.0 PL=0
MOVL C01649 V=800.0 PL=0
MOVL C01650 V=800.0 PL=0
MOVL C01651 V=800.0 PL=0
MOVL C01652 V=800.0 PL=0
MOVL C01653 V=800.0 PL=0
MOVL C01654 V=800.0 PL=0
MOVL C01655 V=800.0 PL=0
MOVL C01656 V=800.0 PL=0
MOVL C01657 V=800.0 PL=0
MOVL C01658 V=800.0 PL=0
MOVL C01659 V=800.0 PL=0
MOVL C01660 V=800.0 PL=0
MOVL C01661 V=800.0 PL=0
MOVL C01662 V=800.0 PL=0
MOVL C01663 V=800.0 PL=0
MOVL C01664 V=800.0 PL=0
MOVL C01665 V=800.0 PL=0
MOVL C01666 V=800.0 PL=0
MOVL C01667 V=800.0 PL=0
MOVL C01668 V=800.0 PL=0
MOVL C01669 V=800.0 PL=0
MOVL C01670 V=800.0 PL=0
MOVL C01671 V=800.0 PL=0
MOVL C01672 V=800.0 PL=0
MOVL C01673 V=800.0 PL=0
MOVL C01674 V=800.0 PL=0
MOVL C01675 V=800.0 PL=0
MOVL C01676 V=800.0 PL=0
MOVL C01677 V=800.0 PL=0
MOVL C01678 V=800.0 PL=0
MOVL C01679 V=800.0 PL=0
MOVL C01680 V=800.0 PL=0
MOVL C01681 V=800.0 PL=0
MOVL C01682 V=800.0 PL=0
MOVL C01683 V=800.0 PL=0
MOVL C01684 V=800.0 PL=0
MOVL C01685 V=800.0 PL=0
MOVL C01686 V=800.0 PL=0
MOVL C01687 V=800.0 PL=0
MOVL C01688 V=800.0 PL=0
MOVL C01689 V=800.0 PL=0
MOVL C01690 V=800.0 PL=0
MOVL C01691 V=800.0 PL=0
MOVL C01692 V=800.0 PL=0
MOVL C01693 V=800.0 PL=0
MOVL C01694 V=800.0 PL=0
MOVL C01695 V=800.0 PL=0
MOVL C01696 V=800.0 PL=0
MOVL C01697 V=800.0 PL=0
MOVL C01698 V=800.0 PL=0
MOVL C01699 V=800.0 PL=0
MOVL C01700 V=800.0 PL=0
MOVL C01701 V=800.0 PL=0
MOVL C01702 V=800.0 PL=0
MOVL C01703 V=800.0 PL=0
MOVL C01704 V=800.0 PL=0
MOVL C01705 V=800.0 PL=0
MOVL C01706 V=800.0 PL=0
MOVL C01707 V=800.0 PL=0
MOVL C01708 V=800.0 PL=0
MOVL C01709 V=800.0 PL=0
MOVL C01710 V=800.0 PL=0
MOVL C01711 V=800.0 PL=0
MOVL C01712 V=800.0 PL=0
MOVL C01713 V=800.0 PL=0
MOVL C01714 V=800.0 PL=0
MOVL C01715 V=800.0 PL=0
MOVL C01716 V=800.0 PL=0
MOVL C01717 V=800.0 PL=0
MOVL C01718 V=800.0 PL=0
MOVL C01719 V=800.0 PL=0
MOVL C01720 V=800.0 PL=0
MOVL C01721 V=800.0 PL=0
MOVL C01722 V=800.0 PL=0
MOVL C01723 V=800.0 PL=0
MOVL C01724 V=800.0 PL=0
MOVL C01725 V=800.0 PL=0
MOVL C01726 V=800.0 PL=0
MOVL C01727 V=800.0 PL=0
MOVL C01728 V=800.0 PL=0
MOVL C01729 V=800.0 PL=0
MOVL C01730 V=800.0 PL=0
MOVL C01731 V=800.0 PL=0
MOVL C01732 V=800.0 PL=0
MOVL C01733 V=800.0 PL=0
MOVL C01734 V=800.0 PL=0
MOVL C01735 V=800.0 PL=0
MOVL C01736 V=800.0 PL=0
MOVL C01737 V=800.0 PL=0
MOVL C01738 V=800.0 PL=0
MOVL C01739 V=800.0 PL=0
MOVL C01740 V=800.0 PL=0
MOVL C01741 V=800.0 PL=0
MOVL C01742 V=800.0 PL=0
MOVL C01743 V=800.0 PL=0
MOVL C01744 V=800.0 PL=0
MOVL C01745 V=800.0 PL=0
MOVL C01746 V=800.0 PL=0
MOVL C01747 V=800.0 PL=0
MOVL C01748 V=800.0 PL=0
MOVL C01749 V=800.0 PL=0
MOVL C01750 V=800.0 PL=0
MOVL C01751 V=800.0 PL=0
MOVL C01752 V=800.0 PL=0
MOVL C01753 V=800.0 PL=0
MOVL C01754 V=800.0 PL=0
MOVL C01755 V=800.0 PL=0
MOVL C01756 V=800.0 PL=0
MOVL C01757 V=800.0 PL=0
MOVL C01758 V=800.0 PL=0
MOVL C01759 V=800.0 PL=0
MOVL C01760 V=800.0 PL=0
MOVL C01761 V=800.0 PL=0
MOVL C01762 V=800.0 PL=0
MOVL C01763 V=800.0 PL=0
MOVL C01764 V=800.0 PL=0
MOVL C01765 V=800.0 PL=0
MOVL C01766 V=800.0 PL=0
MOVL C01767 V=800.0 PL=0
MOVL C01768 V=800.0 PL=0
MOVL C01769 V=800.0 PL=0
MOVL C01770 V=800.0 PL=0
MOVL C01771 V=800.0 PL=0
MOVL C01772 V=800.0 PL=0
MOVL C01773 V=800.0 PL=0
MOVL C01774 V=800.0 PL=0
MOVL C01775 V=800.0 PL=0
MOVL C01776 V=800.0 PL=0
MOVL C01777 V=800.0 PL=0
MOVL C01778 V=800.0 PL=0
MOVL C01779 V=800.0 PL=0
MOVL C01780 V=800.0 PL=0
MOVL C01781 V=800.0 PL=0
MOVL C01782 V=800.0 PL=0
MOVL C01783 V=800.0 PL=0
MOVL C01784 V=800.0 PL=0
MOVL C01785 V=800.0 PL=0
MOVL C01786 V=800.0 PL=0
MOVL C01787 V=800.0 PL=0
MOVL C01788 V=800.0 PL=0
MOVL C01789 V=800.0 PL=0
MOVL C01790 V=800.0 PL=0
MOVL C01791 V=800.0 PL=0
MOVL C01792 V=800.0 PL=0
MOVL C01793 V=800.0 PL=0
MOVL C01794 V=800.0 PL=0
MOVL C01795 V=800.0 PL=0
MOVL C01796 V=800.0 PL=0
MOVL C01797 V=800.0 PL=0
MOVL C01798 V=800.0 PL=0
MOVL C01799 V=800.0 PL=0
MOVL C01800 V=800.0 PL=0
MOVL C01801 V=800.0 PL=0
MOVL C01802 V=800.0 PL=0
MOVL C01803 V=800.0 PL=0
MOVL C01804 V=800.0 PL=0
MOVL C01805 V=800.0 PL=0
MOVL C01806 V=800.0 PL=0
MOVL C01807 V=800.0 PL=0
MOVL C01808 V=800.0 PL=0
MOVL C01809 V=800.0 PL=0
MOVL C01810 V=800.0 PL=0
MOVL C01811 V=800.0 PL=0
MOVL C01812 V=800.0 PL=0
MOVL C01813 V=800.0 PL=0
MOVL C01814 V=800.0 PL=0
MOVL C01815 V=800.0 PL=0
MOVL C01816 V=800.0 PL=0
MOVL C01817 V=800.0 PL=0
MOVL C01818 V=800.0 PL=0
MOVL C01819 V=800.0 PL=0
MOVL C01820 V=800.0 PL=0
MOVL C01821 V=800.0 PL=0
MOVL C01822 V=800.0 PL=0
MOVL C01823 V=800.0 PL=0
MOVL C01824 V=800.0 PL=0
MOVL C01825 V=800.0 PL=0
MOVL C01826 V=800.0 PL=0
MOVL C01827 V=800.0 PL=0
MOVL C01828 V=800.0 PL=0
MOVL C01829 V=800.0 PL=0
MOVL C01830 V=800.0 PL=0
MOVL C01831 V=800.0 PL=0
MOVL C01832 V=800.0 PL=0
MOVL C01833 V=800.0 PL=0
MOVL C01834 V=800.0 PL=0
MOVL C01835 V=800.0 PL=0
MOVL C01836 V=800.0 PL=0
MOVL C01837 V=800.0 PL=0
MOVL C01838 V=800.0 PL=0
MOVL C01839 V=800.0 PL=0
MOVL C01840 V=800.0 PL=0
MOVL C01841 V=800.0 PL=0
MOVL C01842 V=800.0 PL=0
MOVL C01843 V=800.0 PL=0
MOVL C01844 V=800.0 PL=0
MOVL C01845 V=800.0 PL=0
MOVL C01846 V=800.0 PL=0
MOVL C01847 V=800.0 PL=0
MOVL C01848 V=800.0 PL=0
MOVL C01849 V=800.0 PL=0
MOVL C01850 V=800.0 PL=0
MOVL C01851 V=800.0 PL=0
MOVL C01852 V=800.0 PL=0
MOVL C01853 V=800.0 PL=0
MOVL C01854 V=800.0 PL=0
MOVL C01855 V=800.0 PL=0
MOVL C01856 V=800.0 PL=0
MOVL C01857 V=800.0 PL=0
MOVL C01858 V=800.0 PL=0
MOVL C01859 V=800.0 PL=0
MOVL C01860 V=800.0 PL=0
MOVL C01861 V=800.0 PL=0
MOVL C01862 V=800.0 PL=0
MOVL C01863 V=800.0 PL=0
MOVL C01864 V=800.0 PL=0
MOVL C01865 V=800.0 PL=0
MOVL C01866 V=800.0 PL=0
MOVL C01867 V=800.0 PL=0
MOVL C01868 V=800.0 PL=0
MOVL C01869 V=800.0 PL=0
MOVL C01870 V=800.0 PL=0
MOVL C01871 V=800.0 PL=0
MOVL C01872 V=800.0 PL=0
MOVL C01873 V=800.0 PL=0
MOVL C01874 V=800.0 PL=0
MOVL C01875 V=800.0 PL=0
MOVL C01876 V=800.0 PL=0
MOVL C01877 V=800.0 PL=0
MOVL C01878 V=800.0 PL=0
MOVL C01879 V=800.0 PL=0
MOVL C01880 V=800.0 PL=0
MOVL C01881 V=800.0 PL=0
MOVL C01882 V=800.0 PL=0
MOVL C01883 V=800.0 PL=0
MOVL C01884 V=800.0 PL=0
MOVL C01885 V=800.0 PL=0
MOVL C01886 V=800.0 PL=0
MOVL C01887 V=800.0 PL=0
MOVL C01888 V=800.0 PL=0
MOVL C01889 V=800.0 PL=0
MOVL C01890 V=800.0 PL=0
MOVL C01891 V=800.0 PL=0
MOVL C01892 V=800.0 PL=0
MOVL C01893 V=800.0 PL=0
MOVL C01894 V=800.0 PL=0
MOVL C01895 V=800.0 PL=0
MOVL C01896 V=800.0 PL=0
MOVL C01897 V=800.0 PL=0
MOVL C01898 V=800.0 PL=0
MOVL C01899 V=800.0 PL=0
MOVL C01900 V=800.0 PL=0
MOVL C01901 V=800.0 PL=0
MOVL C01902 V=800.0 PL=0
MOVL C01903 V=800.0 PL=0
MOVL C01904 V=800.0 PL=0
MOVL C01905 V=800.0 PL=0
MOVL C01906 V=800.0 PL=0
MOVL C01907 V=800.0 PL=0
MOVL C01908 V=800.0 PL=0
MOVL C01909 V=800.0 PL=0
MOVL C01910 V=800.0 PL=0
MOVL C01911 V=800.0 PL=0
MOVL C01912 V=800.0 PL=0
MOVL C01913 V=800.0 PL=0
MOVL C01914 V=800.0 PL=0
MOVL C01915 V=800.0 PL=0
MOVL C01916 V=800.0 PL=0
MOVL C01917 V=800.0 PL=0
MOVL C01918 V=800.0 PL=0
MOVL C01919 V=800.0 PL=0
MOVL C01920 V=800.0 PL=0
MOVL C01921 V=800.0 PL=0
MOVL C01922 V=800.0 PL=0
MOVL C01923 V=800.0 PL=0
MOVL C01924 V=800.0 PL=0
MOVL C01925 V=800.0 PL=0
MOVL C01926 V=800.0 PL=0
MOVL C01927 V=800.0 PL=0
MOVL C01928 V=800.0 PL=0
MOVL C01929 V=800.0 PL=0
MOVL C01930 V=800.0 PL=0
MOVL C01931 V=800.0 PL=0
MOVL C01932 V=800.0 PL=0
MOVL C01933 V=800.0 PL=0
MOVL C01934 V=800.0 PL=0
MOVL C01935 V=800.0 PL=0
MOVL C01936 V=800.0 PL=0
MOVL C01937 V=800.0 PL=0
MOVL C01938 V=800.0 PL=0
MOVL C01939 V=800.0 PL=0
MOVL C01940 V=800.0 PL=0
MOVL C01941 V=800.0 PL=0
MOVL C01942 V=800.0 PL=0
MOVL C01943 V=800.0 PL=0
MOVL C01944 V=800.0 PL=0
MOVL C01945 V=800.0 PL=0
MOVL C01946 V=800.0 PL=0
MOVL C01947 V=800.0 PL=0
MOVL C01948 V=800.0 PL=0
MOVL C01949 V=800.0 PL=0
MOVL C01950 V=800.0 PL=0
MOVL C01951 V=800.0 PL=0
MOVL C01952 V=800.0 PL=0
MOVL C01953 V=800.0 PL=0
MOVL C01954 V=800.0 PL=0
MOVL C01955 V=800.0 PL=0
MOVL C01956 V=800.0 PL=0
MOVL C01957 V=800.0 PL=0
MOVL C01958 V=800.0 PL=0
MOVL C01959 V=800.0 PL=0
MOVL C01960 V=800.0 PL=0
MOVL C01961 V=800.0 PL=0
MOVL C01962 V=800.0 PL=0
MOVL C01963 V=800.0 PL=0
MOVL C01964 V=800.0 PL=0
MOVL C01965 V=800.0 PL=0
MOVL C01966 V=800.0 PL=0
MOVL C01967 V=800.0 PL=0
MOVL C01968 V=800.0 PL=0
MOVL C01969 V=800.0 PL=0
MOVL C01970 V=800.0 PL=0
MOVL C01971 V=800.0 PL=0
MOVL C01972 V=800.0 PL=0
MOVL C01973 V=800.0 PL=0
MOVL C01974 V=800.0 PL=0
MOVL C01975 V=800.0 PL=0
MOVL C01976 V=800.0 PL=0
MOVL C01977 V=800.0 PL=0
MOVL C01978 V=800.0 PL=0
MOVL C01979 V=800.0 PL=0
MOVL C01980 V=800.0 PL=0
MOVL C01981 V=800.0 PL=0
MOVL C01982 V=800.0 PL=0
MOVL C01983 V=800.0 PL=0
MOVL C01984 V=800.0 PL=0
MOVL C01985 V=800.0 PL=0
MOVL C01986 V=800.0 PL=0
MOVL C01987 V=800.0 PL=0
MOVL C01988 V=800.0 PL=0
MOVL C01989 V=800.0 PL=0
MOVL C01990 V=800.0 PL=0
MOVL C01991 V=800.0 PL=0
MOVL C01992 V=800.0 PL=0
MOVL C01993 V=800.0 PL=0
MOVL C01994 V=800.0 PL=0
MOVL C01995 V=800.0 PL=0
MOVL C01996 V=800.0 PL=0
MOVL C01997 V=800.0 PL=0
MOVL C01998 V=800.0 PL=0
MOVL C01999 V=800.0 PL=0
MOVL C02000 V=800.0 PL=0
MOVL C02001 V=800.0 PL=0
MOVL C02002 V=800.0 PL=0
MOVL C02003 V=800.0 PL=0
MOVL C02004 V=800.0 PL=0
MOVL C02005 V=800.0 PL=0
MOVL C02006 V=800.0 PL=0
MOVL C02007 V=800.0 PL=0
MOVL C02008 V=800.0 PL=0
MOVL C02009 V=800.0 PL=0
MOVL C02010 V=800.0 PL=0
MOVL C02011 V=800.0 PL=0
MOVL C02012 V=800.0 PL=0
MOVL C02013 V=800.0 PL=0
MOVL C02014 V=800.0 PL=0
MOVL C02015 V=800.0 PL=0
MOVL C02016 V=800.0 PL=0
MOVL C02017 V=800.0 PL=0
MOVL C02018 V=800.0 PL=0
MOVL C02019 V=800.0 PL=0
MOVL C02020 V=800.0 PL=0
MOVL C02021 V=800.0 PL=0
MOVL C02022 V=800.0 PL=0
MOVL C02023 V=800.0 PL=0
MOVL C02024 V=800.0 PL=0
MOVL C02025 V=800.0 PL=0
MOVL C02026 V=800.0 PL=0
MOVL C02027 V=800.0 PL=0
MOVL C02028 V=800.0 PL=0
MOVL C02029 V=800.0 PL=0
MOVL C02030 V=800.0 PL=0
MOVL C02031 V=800.0 PL=0
MOVL C02032 V=800.0 PL=0
MOVL C02033 V=800.0 PL=0
MOVL C02034 V=800.0 PL=0
MOVL C02035 V=800.0 PL=0
MOVL C02036 V=800.0 PL=0
MOVL C02037 V=800.0 PL=0
MOVL C02038 V=800.0 PL=0
MOVL C02039 V=800.0 PL=0
MOVL C02040 V=800.0 PL=0
MOVL C02041 V=800.0 PL=0
MOVL C02042 V=800.0 PL=0
MOVL C02043 V=800.0 PL=0
MOVL C02044 V=800.0 PL=0
MOVL C02045 V=800.0 PL=0
MOVL C02046 V=800.0 PL=0
MOVL C02047 V=800.0 PL=0
MOVL C02048 V=800.0 PL=0
MOVL C02049 V=800.0 PL=0
MOVL C02050 V=800.0 PL=0
MOVL C02051 V=800.0 PL=0
MOVL C02052 V=800.0 PL=0
MOVL C02053 V=800.0 PL=0
MOVL C02054 V=800.0 PL=0
MOVL C02055 V=800.0 PL=0
MOVL C02056 V=800.0 PL=0
MOVL C02057 V=800.0 PL=0
MOVL C02058 V=800.0 PL=0
MOVL C02059 V=800.0 PL=0
MOVL C02060 V=800.0 PL=0
MOVL C02061 V=800.0 PL=0
MOVL C02062 V=800.0 PL=0
MOVL C02063 V=800.0 PL=0
MOVL C02064 V=800.0 PL=0
MOVL C02065 V=800.0 PL=0
MOVL C02066 V=800.0 PL=0
MOVL C02067 V=800.0 PL=0
MOVL C02068 V=800.0 PL=0
MOVL C02069 V=800.0 PL=0
MOVL C02070 V=800.0 PL=0
MOVL C02071 V=800.0 PL=0
MOVL C02072 V=800.0 PL=0
MOVL C02073 V=800.0 PL=0
MOVL C02074 V=800.0 PL=0
MOVL C02075 V=800.0 PL=0
MOVL C02076 V=800.0 PL=0
MOVL C02077 V=800.0 PL=0
MOVL C02078 V=800.0 PL=0
MOVL C02079 V=800.0 PL=0
MOVL C02080 V=800.0 PL=0
MOVL C02081 V=800.0 PL=0
MOVL C02082 V=800.0 PL=0
MOVL C02083 V=800.0 PL=0
MOVL C02084 V=800.0 PL=0
MOVL C02085 V=800.0 PL=0
MOVL C02086 V=800.0 PL=0
MOVL C02087 V=800.0 PL=0
MOVL C02088 V=800.0 PL=0
MOVL C02089 V=800.0 PL=0
MOVL C02090 V=800.0 PL=0
MOVL C02091 V=800.0 PL=0
MOVL C02092 V=800.0 PL=0
MOVL C02093 V=800.0 PL=0
MOVL C02094 V=800.0 PL=0
MOVL C02095 V=800.0 PL=0
MOVL C02096 V=800.0 PL=0
MOVL C02097 V=800.0 PL=0
MOVL C02098 V=800.0 PL=0
MOVL C02099 V=800.0 PL=0
MOVL C02100 V=800.0 PL=0
MOVL C02101 V=800.0 PL=0
MOVL C02102 V=800.0 PL=0
MOVL C02103 V=800.0 PL=0
MOVL C02104 V=800.0 PL=0
MOVL C02105 V=800.0 PL=0
MOVL C02106 V=800.0 PL=0
MOVL C02107 V=800.0 PL=0
MOVL C02108 V=800.0 PL=0
MOVL C02109 V=800.0 PL=0
MOVL C02110 V=800.0 PL=0
MOVL C02111 V=800.0 PL=0
MOVL C02112 V=800.0 PL=0
MOVL C02113 V=800.0 PL=0
MOVL C02114 V=800.0 PL=0
MOVL C02115 V=800.0 PL=0
MOVL C02116 V=800.0 PL=0
MOVL C02117 V=800.0 PL=0
MOVL C02118 V=800.0 PL=0
MOVL C02119 V=800.0 PL=0
MOVL C02120 V=800.0 PL=0
MOVL C02121 V=800.0 PL=0
MOVL C02122 V=800.0 PL=0
MOVL C02123 V=800.0 PL=0
MOVL C02124 V=800.0 PL=0
MOVL C02125 V=800.0 PL=0
MOVL C02126 V=800.0 PL=0
MOVL C02127 V=800.0 PL=0
MOVL C02128 V=800.0 PL=0
MOVL C02129 V=800.0 PL=0
MOVL C02130 V=800.0 PL=0
MOVL C02131 V=800.0 PL=0
MOVL C02132 V=800.0 PL=0
MOVL C02133 V=800.0 PL=0
MOVL C02134 V=800.0 PL=0
MOVL C02135 V=800.0 PL=0
MOVL C02136 V=800.0 PL=0
MOVL C02137 V=800.0 PL=0
MOVL C02138 V=800.0 PL=0
MOVL C02139 V=800.0 PL=0
MOVL C02140 V=800.0 PL=0
MOVL C02141 V=800.0 PL=0
MOVL C02142 V=800.0 PL=0
MOVL C02143 V=800.0 PL=0
